DATA_BLOCK "DB_RecordData"   // DB70
{ S7_Optimized_Access := 'TRUE' }
// stored: AutoNumber false, MemoryReserve 100
   VAR
      xFP_ExportProdData { ExternalAccessible := 'False'; ExternalVisible := 'False'; ExternalWritable := 'False'} : Bool;
      xFP_ExportFlatCtrlRobot1 { ExternalAccessible := 'False'; ExternalVisible := 'False'; ExternalWritable := 'False'} : Bool;
      xFP_ExportFlatCtrlRobot2 { ExternalAccessible := 'False'; ExternalVisible := 'False'; ExternalWritable := 'False'} : Bool;
      xWriteDblExportProdDataBusy { ExternalAccessible := 'False'; ExternalVisible := 'False'; ExternalWritable := 'False'} : Bool;
      xWriteDblExportflatCtrlR1Busy { ExternalAccessible := 'False'; ExternalVisible := 'False'; ExternalWritable := 'False'} : Bool;
      xWriteDblExportFlatCtrlR2Busy { ExternalAccessible := 'False'; ExternalVisible := 'False'; ExternalWritable := 'False'} : Bool;
      nWriteDblExportProdDataResult { ExternalAccessible := 'False'; ExternalVisible := 'False'; ExternalWritable := 'False'} : Int;
      nWriteDblExportflatCtrlR1Result { ExternalAccessible := 'False'; ExternalVisible := 'False'; ExternalWritable := 'False'} : Int;
      nWriteDblExportFlatCtrlR2Result { ExternalAccessible := 'False'; ExternalVisible := 'False'; ExternalWritable := 'False'} : Int;
      xExportProdDataDone { ExternalAccessible := 'False'; ExternalVisible := 'False'; ExternalWritable := 'False'} : Bool;
      xExportProdDataBusy { ExternalAccessible := 'False'; ExternalVisible := 'False'; ExternalWritable := 'False'} : Bool;
      xExportProdDataError { ExternalAccessible := 'False'; ExternalVisible := 'False'; ExternalWritable := 'False'} : Bool;
      wExportProdDataStatus { ExternalAccessible := 'False'; ExternalVisible := 'False'; ExternalWritable := 'False'} : Word;
      wMemExportProdDataStatus { ExternalAccessible := 'False'; ExternalVisible := 'False'; ExternalWritable := 'False'} : Word;
      xExportFlatCtrlR1Done { ExternalAccessible := 'False'; ExternalVisible := 'False'; ExternalWritable := 'False'} : Bool;
      xExportFlatCtrlR1Busy { ExternalAccessible := 'False'; ExternalVisible := 'False'; ExternalWritable := 'False'} : Bool;
      xExportFlatCtrlR1Error { ExternalAccessible := 'False'; ExternalVisible := 'False'; ExternalWritable := 'False'} : Bool;
      wExportFlatCtrlR1Status { ExternalAccessible := 'False'; ExternalVisible := 'False'; ExternalWritable := 'False'} : Word;
      wMemExportFlatCtrlR1Status { ExternalAccessible := 'False'; ExternalVisible := 'False'; ExternalWritable := 'False'} : Word;
      xExportFlatCtrlR2Done { ExternalAccessible := 'False'; ExternalVisible := 'False'; ExternalWritable := 'False'} : Bool;
      xExportFlatCtrlR2Busy { ExternalAccessible := 'False'; ExternalVisible := 'False'; ExternalWritable := 'False'} : Bool;
      xExportFlatCtrlR2Error { ExternalAccessible := 'False'; ExternalVisible := 'False'; ExternalWritable := 'False'} : Bool;
      wExportFlatCtrlR2Status { ExternalAccessible := 'False'; ExternalVisible := 'False'; ExternalWritable := 'False'} : Word;
      wMemExportFlatCtrlR2Status { ExternalAccessible := 'False'; ExternalVisible := 'False'; ExternalWritable := 'False'} : Word;
   END_VAR
BEGIN
END_DATA_BLOCK

DATA_BLOCK "DBF_Safety"   // DB901, F_DB
{ S7_Optimized_Access := 'TRUE' }
// stored: AutoNumber false
   VAR
      TrueSafety { ExternalAccessible := 'False'; ExternalVisible := 'False'; ExternalWritable := 'False'} : Bool := TRUE;   // Safety Bool always TRUE
      FalseSafety { ExternalAccessible := 'False'; ExternalVisible := 'False'; ExternalWritable := 'False'} : Bool := FALSE;   // Safety Bool always FALSE
      Reset { ExternalAccessible := 'False'; ExternalVisible := 'False'; ExternalWritable := 'False'} : Bool;   // Reset bool
      ResetDoor { ExternalAccessible := 'False'; ExternalVisible := 'False'; ExternalWritable := 'False'} : Bool;   // Reset bool on maintenance door acces
      i_EStopOnMainCabinet { ExternalAccessible := 'False'; ExternalVisible := 'False'; ExternalWritable := 'False'} : Bool;   // Emergency stop state on main cabinet
      i_EStopLeftRopePull { ExternalAccessible := 'False'; ExternalVisible := 'False'; ExternalWritable := 'False'} : Bool;   // Emergency stop state rope pull left
      i_EStopRightRopePull { ExternalAccessible := 'False'; ExternalVisible := 'False'; ExternalWritable := 'False'} : Bool;   // Emergency stop state rope full right
      i_EStopEntryDoor { ExternalAccessible := 'False'; ExternalVisible := 'False'; ExternalWritable := 'False'} : Bool;   // Emergency stop state on entry guard locking
      i_DoorAcces { ExternalAccessible := 'False'; ExternalVisible := 'False'; ExternalWritable := 'False'} : Bool;   // Door state
      i_GateAccesCBS { ExternalAccessible := 'False'; ExternalVisible := 'False'; ExternalWritable := 'False'} : Bool;   // Gate acces state
      i_EStopControlRoom { ExternalAccessible := 'False'; ExternalVisible := 'False'; ExternalWritable := 'False'} : Bool;   // Emergency stop in the control room
      i_PedestrialDoorAcces { ExternalAccessible := 'False'; ExternalVisible := 'False'; ExternalWritable := 'False'} : Bool;   // Pedestrial door access state
      i_CaptiveKeyInLock { ExternalAccessible := 'False'; ExternalVisible := 'False'; ExternalWritable := 'False'} : Bool;   // Captive key on Lock
      i_EStopFromLeftRobot { ExternalAccessible := 'False'; ExternalVisible := 'False'; ExternalWritable := 'False'} : Bool;   // Emergency stop from flex pendant on the left robot
      i_EStopFromRightRobot { ExternalAccessible := 'False'; ExternalVisible := 'False'; ExternalWritable := 'False'} : Bool;   // Emergency stop from flex pendant on the right robot
      i_ReqEnableAirLeft { ExternalAccessible := 'False'; ExternalVisible := 'False'; ExternalWritable := 'False'} : Bool;   // Request enavle air pressure supply from left robot
      i_ReqEnableAirRight { ExternalAccessible := 'False'; ExternalVisible := 'False'; ExternalWritable := 'False'} : Bool;   // Request enavle air pressure supply from right robot
      i_RobotLeftStopped { ExternalAccessible := 'False'; ExternalVisible := 'False'; ExternalWritable := 'False'} : Bool;   // Left robot stooped
      i_RobotRightStopped { ExternalAccessible := 'False'; ExternalVisible := 'False'; ExternalWritable := 'False'} : Bool;   // Right robot stopped
      i_VacuumPumpRunning { ExternalAccessible := 'False'; ExternalVisible := 'False'; ExternalWritable := 'False'} : Bool;
      o_EnableAirSupplyLeftRobot { ExternalAccessible := 'False'; ExternalVisible := 'False'; ExternalWritable := 'False'} : Bool;   // Enable air pressure supply for left robot
      o_EnableAirSupplyRightRobot { ExternalAccessible := 'False'; ExternalVisible := 'False'; ExternalWritable := 'False'} : Bool;   // Enable air pressure supply for right robot
      o_EnableAirSupplySuctionUnit { ExternalAccessible := 'False'; ExternalVisible := 'False'; ExternalWritable := 'False'} : Bool;   // Enable air pressure supply for suction unit
      o_EStopSuctionUnit { ExternalAccessible := 'False'; ExternalVisible := 'False'; ExternalWritable := 'False'} : Bool;   // Emergency stop state to suction unit
      o_EStopToLeftRobot { ExternalAccessible := 'False'; ExternalVisible := 'False'; ExternalWritable := 'False'} : Bool;   // Cell emergency stop to left robot
      o_EStopToRightRobot { ExternalAccessible := 'False'; ExternalVisible := 'False'; ExternalWritable := 'False'} : Bool;   // Cell emergency stop to right robot
      o_OperatorProtectionToLeftRobot { ExternalAccessible := 'False'; ExternalVisible := 'False'; ExternalWritable := 'False'} : Bool;   // Operator protection state to the left robot
      o_OperatorProtectionToRightRobot { ExternalAccessible := 'False'; ExternalVisible := 'False'; ExternalWritable := 'False'} : Bool;   // Operator protection state to the right robot
      o_VacuumRunningDelayed { ExternalAccessible := 'False'; ExternalVisible := 'False'; ExternalWritable := 'False'} : Bool;   // Vacuum running delayed of
      l_GlobalEmergencyStopCell { ExternalAccessible := 'False'; ExternalVisible := 'False'; ExternalWritable := 'False'} : Bool;   // Global Emergency stop cell state
      l_GlobalEmergencyStop { ExternalAccessible := 'False'; ExternalVisible := 'False'; ExternalWritable := 'False'} : Bool;   // Global Emergency stop state
      l_GlobalEStopToLeftRobot { ExternalAccessible := 'False'; ExternalVisible := 'False'; ExternalWritable := 'False'} : Bool;   // Global Emergency stop state send to left robot
      l_GlobalEStopToRightRobot { ExternalAccessible := 'False'; ExternalVisible := 'False'; ExternalWritable := 'False'} : Bool;   // Global Emergency stop state send to right robot
      l_GlobalOperatorProtection { ExternalAccessible := 'False'; ExternalVisible := 'False'; ExternalWritable := 'False'} : Bool;   // Global door and gate state
      xErrorReadFromLeft { ExternalAccessible := 'False'; ExternalVisible := 'False'; ExternalWritable := 'False'} : Bool;
      xErrorReadFromRight { ExternalAccessible := 'False'; ExternalVisible := 'False'; ExternalWritable := 'False'} : Bool;
      xErrorWriteToLeft { ExternalAccessible := 'False'; ExternalVisible := 'False'; ExternalWritable := 'False'} : Bool;
      xErrorWriteToRight { ExternalAccessible := 'False'; ExternalVisible := 'False'; ExternalWritable := 'False'} : Bool;
      xAuthorStart { ExternalAccessible := 'False'; ExternalVisible := 'False'; ExternalWritable := 'False'} : Bool;
      xVacuumPumpRunning { ExternalAccessible := 'False'; ExternalVisible := 'False'; ExternalWritable := 'False'} : Bool;
   END_VAR
BEGIN
END_DATA_BLOCK

DATA_BLOCK "DB_FromSafety"   // DB998
{ S7_Optimized_Access := 'TRUE' }
// stored: AutoNumber false, MemoryReserve 100
   VAR
      EStopOnMainCabinet { ExternalAccessible := 'False'; ExternalVisible := 'False'; ExternalWritable := 'False'} : "stSafetyState";
      EstopLeftRopePull { ExternalAccessible := 'False'; ExternalVisible := 'False'; ExternalWritable := 'False'} : "stSafetyState";
      EstopRightRopePull { ExternalAccessible := 'False'; ExternalVisible := 'False'; ExternalWritable := 'False'} : "stSafetyState";
      EStopEntryDoor { ExternalAccessible := 'False'; ExternalVisible := 'False'; ExternalWritable := 'False'} : "stSafetyState";
      DoorAcces { ExternalAccessible := 'False'; ExternalVisible := 'False'; ExternalWritable := 'False'} : "stSafetyState";
      GateAccesCBS { ExternalAccessible := 'False'; ExternalVisible := 'False'; ExternalWritable := 'False'} : "stSafetyState";
      EStopControlRoom { ExternalAccessible := 'False'; ExternalVisible := 'False'; ExternalWritable := 'False'} : "stSafetyState";
      EnableAirSupplyLeftRobot { ExternalAccessible := 'False'; ExternalVisible := 'False'; ExternalWritable := 'False'} : "stSafetyState";
      EnableAirSupplyRightRobot { ExternalAccessible := 'False'; ExternalVisible := 'False'; ExternalWritable := 'False'} : "stSafetyState";
      EnableAirSupplySuctionUnit { ExternalAccessible := 'False'; ExternalVisible := 'False'; ExternalWritable := 'False'} : "stSafetyState";
      EStopSuctionUnit { ExternalAccessible := 'False'; ExternalVisible := 'False'; ExternalWritable := 'False'} : "stSafetyState";
      PedestrialDoorAcces { ExternalAccessible := 'False'; ExternalVisible := 'False'; ExternalWritable := 'False'} : "stSafetyState";
      CaptiveKeyInLock { ExternalAccessible := 'False'; ExternalVisible := 'False'; ExternalWritable := 'False'} : "stSafetyState";
      VacuumPumpRunning { ExternalAccessible := 'False'; ExternalVisible := 'False'; ExternalWritable := 'False'} : "stSafetyState";
      GlobalEStop { ExternalAccessible := 'False'; ExternalVisible := 'False'; ExternalWritable := 'False'; S7_SetPoint := 'True'} : "stSafetyState";
      xLeftRobotStopped { ExternalAccessible := 'False'; ExternalVisible := 'False'; ExternalWritable := 'False'} : Bool;
      xRightRobotStopped { ExternalAccessible := 'False'; ExternalVisible := 'False'; ExternalWritable := 'False'} : Bool;
      xEStopLeftRobot { ExternalAccessible := 'False'; ExternalVisible := 'False'; ExternalWritable := 'False'} : Bool;
      xEStopRightRobot { ExternalAccessible := 'False'; ExternalVisible := 'False'; ExternalWritable := 'False'} : Bool;
      xGlobalSafetyLeft { ExternalAccessible := 'False'; ExternalVisible := 'False'; ExternalWritable := 'False'} : Bool;
      xGlobalSafetyRight { ExternalAccessible := 'False'; ExternalVisible := 'False'; ExternalWritable := 'False'} : Bool;
      xAuthorStartVacuum { ExternalAccessible := 'False'; ExternalVisible := 'False'; ExternalWritable := 'False'} : Bool;
   END_VAR
BEGIN
END_DATA_BLOCK

DATA_BLOCK "DB_ToSafety"   // DB999
{ S7_Optimized_Access := 'TRUE' }
// stored: AutoNumber false, MemoryReserve 100
   VAR
      Reset { ExternalAccessible := 'False'; ExternalVisible := 'False'; ExternalWritable := 'False'} : Bool;   // Commande reset general
      ResetDoor { ExternalAccessible := 'False'; ExternalVisible := 'False'; ExternalWritable := 'False'} : Bool;   // Commande reset porte d'acces maintenance
      DoorLocked { ExternalAccessible := 'False'; ExternalVisible := 'False'; ExternalWritable := 'False'} : Bool;   // The door was locked
      VacuumDriveRunning { ExternalAccessible := 'False'; ExternalVisible := 'False'; ExternalWritable := 'False'} : Bool;   // Vacuum drive is running
      EnableVacuumRunning { ExternalAccessible := 'False'; ExternalVisible := 'False'; ExternalWritable := 'False'} : Bool;   // Enable vacuum running
   END_VAR
BEGIN
END_DATA_BLOCK

ORGANIZATION_BLOCK "Main"   // OB1, LAD, ProgramCycle
TITLE = "Main Program Sweep (Cycle)"
{ S7_Optimized_Access := 'TRUE' }
// stored: SetENOAutomatically false
   VAR_INPUT
      Initial_Call : Bool;   // Initial call of this OB
      Remanence : Bool;   // =True, if remanent data are available
   END_VAR
BEGIN

REGION Network 1
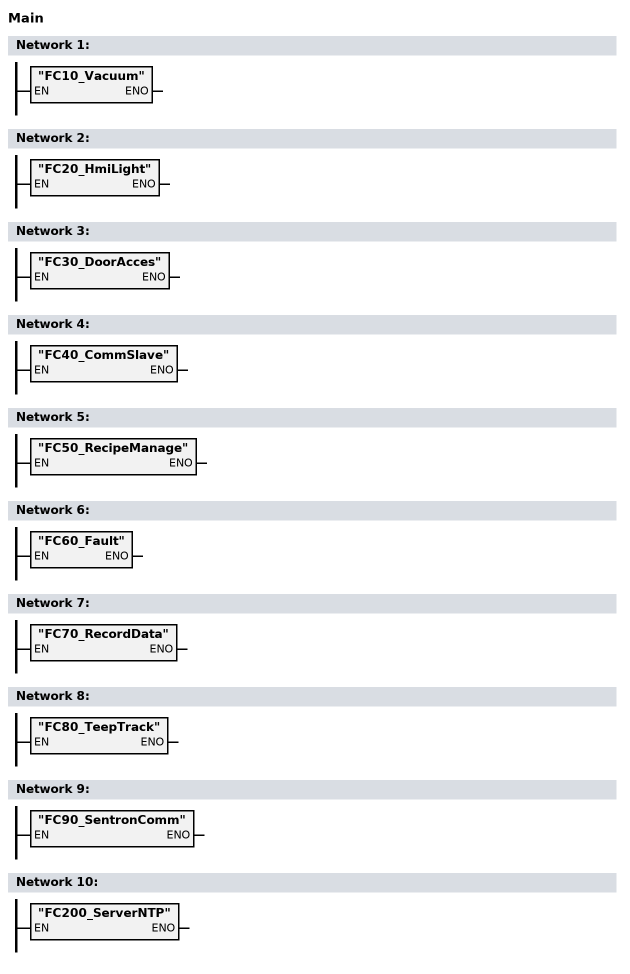
   RUNG wire#powerrail
      "FC10_Vacuum"()
   END_RUNG
   // the same network as SCL:
   "FC10_Vacuum"();
END_REGION

REGION Network 2
   RUNG wire#powerrail
      "FC20_HmiLight"()
   END_RUNG
   // the same network as SCL:
   "FC20_HmiLight"();
END_REGION

REGION Network 3
   RUNG wire#powerrail
      "FC30_DoorAcces"()
   END_RUNG
   // the same network as SCL:
   "FC30_DoorAcces"();
END_REGION

REGION Network 4
   RUNG wire#powerrail
      "FC40_CommSlave"()
   END_RUNG
   // the same network as SCL:
   "FC40_CommSlave"();
END_REGION

REGION Network 5
   RUNG wire#powerrail
      "FC50_RecipeManage"()
   END_RUNG
   // the same network as SCL:
   "FC50_RecipeManage"();
END_REGION

REGION Network 6
   RUNG wire#powerrail
      "FC60_Fault"()
   END_RUNG
   // the same network as SCL:
   "FC60_Fault"();
END_REGION

REGION Network 7
   RUNG wire#powerrail
      "FC70_RecordData"()
   END_RUNG
   // the same network as SCL:
   "FC70_RecordData"();
END_REGION

REGION Network 8
   RUNG wire#powerrail
      "FC80_TeepTrack"()
   END_RUNG
   // the same network as SCL:
   "FC80_TeepTrack"();
END_REGION

REGION Network 9
   RUNG wire#powerrail
      "FC90_SentronComm"()
   END_RUNG
   // the same network as SCL:
   "FC90_SentronComm"();
END_REGION

REGION Network 10
   RUNG wire#powerrail
      "FC200_ServerNTP"()
   END_RUNG
   // the same network as SCL:
   "FC200_ServerNTP"();
END_REGION
END_ORGANIZATION_BLOCK

FUNCTION "FC10_Vacuum" : Void   // FC10, LAD
{ S7_Optimized_Access := 'TRUE' }
// stored: AutoNumber false, IsIECCheckEnabled true, SetENOAutomatically false
BEGIN

REGION Network 1: Complet management of Vacuum system
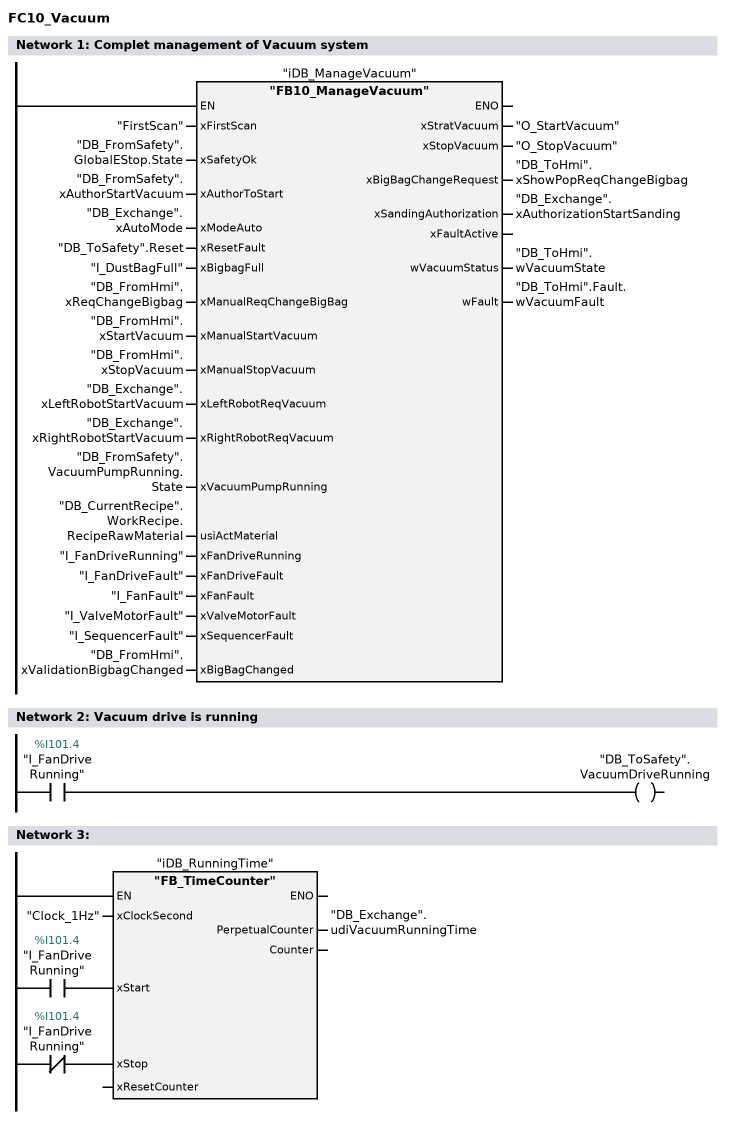
   RUNG wire#powerrail
      "iDB_ManageVacuum"(xFirstScan := "FirstScan", xSafetyOk := "DB_FromSafety".GlobalEStop.State, xAuthorToStart := "DB_FromSafety".xAuthorStartVacuum, xModeAuto := "DB_Exchange".xAutoMode, xResetFault := "DB_ToSafety".Reset, xBigbagFull := "I_DustBagFull", xManualReqChangeBigBag := "DB_FromHmi".xReqChangeBigbag, xManualStartVacuum := "DB_FromHmi".xStartVacuum, xManualStopVacuum := "DB_FromHmi".xStopVacuum, xLeftRobotReqVacuum := "DB_Exchange".xLeftRobotStartVacuum, xRightRobotReqVacuum := "DB_Exchange".xRightRobotStartVacuum, xVacuumPumpRunning := "DB_FromSafety".VacuumPumpRunning.State, usiActMaterial := "DB_CurrentRecipe".WorkRecipe.RecipeRawMaterial, xFanDriveRunning := "I_FanDriveRunning", xFanDriveFault := "I_FanDriveFault", xFanFault := "I_FanFault", xValveMotorFault := "I_ValveMotorFault", xSequencerFault := "I_SequencerFault", xBigBagChanged := "DB_FromHmi".xValidationBigbagChanged, xStratVacuum => "O_StartVacuum", xStopVacuum => "O_StopVacuum", xBigBagChangeRequest => "DB_ToHmi".xShowPopReqChangeBigbag, xSandingAuthorization => "DB_Exchange".xAuthorizationStartSanding, xFaultActive =>, wVacuumStatus => "DB_ToHmi".wVacuumState, wFault => "DB_ToHmi".Fault.wVacuumFault)
   END_RUNG
   // the same network as SCL:
   "iDB_ManageVacuum"(xFirstScan := "FirstScan",   // "FB10_ManageVacuum"
                      xSafetyOk := "DB_FromSafety".GlobalEStop.State,
                      xAuthorToStart := "DB_FromSafety".xAuthorStartVacuum,
                      xModeAuto := "DB_Exchange".xAutoMode,
                      xResetFault := "DB_ToSafety".Reset,
                      xBigbagFull := "I_DustBagFull",
                      xManualReqChangeBigBag := "DB_FromHmi".xReqChangeBigbag,
                      xManualStartVacuum := "DB_FromHmi".xStartVacuum,
                      xManualStopVacuum := "DB_FromHmi".xStopVacuum,
                      xLeftRobotReqVacuum := "DB_Exchange".xLeftRobotStartVacuum,
                      xRightRobotReqVacuum := "DB_Exchange".xRightRobotStartVacuum,
                      xVacuumPumpRunning := "DB_FromSafety".VacuumPumpRunning.State,
                      usiActMaterial := "DB_CurrentRecipe".WorkRecipe.RecipeRawMaterial,
                      xFanDriveRunning := "I_FanDriveRunning",
                      xFanDriveFault := "I_FanDriveFault",
                      xFanFault := "I_FanFault",
                      xValveMotorFault := "I_ValveMotorFault",
                      xSequencerFault := "I_SequencerFault",
                      xBigBagChanged := "DB_FromHmi".xValidationBigbagChanged,
                      xStratVacuum => "O_StartVacuum",
                      xStopVacuum => "O_StopVacuum",
                      xBigBagChangeRequest => "DB_ToHmi".xShowPopReqChangeBigbag,
                      xSandingAuthorization => "DB_Exchange".xAuthorizationStartSanding,
                      wVacuumStatus => "DB_ToHmi".wVacuumState,
                      wFault => "DB_ToHmi".Fault.wVacuumFault);
END_REGION

REGION Network 2: Vacuum drive is running
   RUNG wire#powerrail
      Contact( "I_FanDriveRunning" )
      Coil( "DB_ToSafety".VacuumDriveRunning )
   END_RUNG
   // the same network as SCL:
   "DB_ToSafety".VacuumDriveRunning := "I_FanDriveRunning";
END_REGION

REGION Network 3
   RUNG wire#powerrail
      "iDB_RunningTime"(xStart := wire#w1, xStop := wire#w2, xClockSecond := "Clock_1Hz", xResetCounter :=, PerpetualCounter => "DB_Exchange".udiVacuumRunningTime, "Counter" =>)
   END_RUNG
   RUNG wire#powerrail
      Contact( "I_FanDriveRunning" )
   END_RUNG wire#w1
   RUNG wire#powerrail
      I_Contact( "I_FanDriveRunning" )
   END_RUNG wire#w2
   // the same network as SCL:
   "iDB_RunningTime"(xClockSecond := "Clock_1Hz",   // "FB_TimeCounter"
                     xStart := "I_FanDriveRunning",
                     xStop := NOT "I_FanDriveRunning",
                     PerpetualCounter => "DB_Exchange".udiVacuumRunningTime);
END_REGION
END_FUNCTION

FUNCTION_BLOCK "FB10_ManageVacuum"   // FB10, LAD
{ S7_Optimized_Access := 'TRUE' }
// stored: AutoNumber false, IsIECCheckEnabled true, MemoryReserve 100, SetENOAutomatically true
   VAR_INPUT
      xFirstScan { ExternalAccessible := 'False'; ExternalVisible := 'False'; ExternalWritable := 'False'} : Bool;
      xSafetyOk { ExternalAccessible := 'False'; ExternalVisible := 'False'; ExternalWritable := 'False'} : Bool;   // General Safety state
      xAuthorToStart { ExternalAccessible := 'False'; ExternalVisible := 'False'; ExternalWritable := 'False'} : Bool;   // Authorisation to start Vacuum
      xModeAuto { ExternalAccessible := 'False'; ExternalVisible := 'False'; ExternalWritable := 'False'} : Bool;   // Mode auto active
      xResetFault { ExternalAccessible := 'False'; ExternalVisible := 'False'; ExternalWritable := 'False'} : Bool;   // Reset fault
      xBigbagFull { ExternalAccessible := 'False'; ExternalVisible := 'False'; ExternalWritable := 'False'} : Bool;   // Big Bag is full
      xManualReqChangeBigBag { ExternalAccessible := 'False'; ExternalVisible := 'False'; ExternalWritable := 'False'} : Bool;   // Manual request changing Big bag
      xManualStartVacuum { ExternalAccessible := 'False'; ExternalVisible := 'False'; ExternalWritable := 'False'} : Bool;   // Manual enabling Vacuum
      xManualStopVacuum { ExternalAccessible := 'False'; ExternalVisible := 'False'; ExternalWritable := 'False'} : Bool;   // Manual stopping Vacuum
      xLeftRobotReqVacuum { ExternalAccessible := 'False'; ExternalVisible := 'False'; ExternalWritable := 'False'} : Bool;   // Left Robot request enabling Vacuum
      xRightRobotReqVacuum { ExternalAccessible := 'False'; ExternalVisible := 'False'; ExternalWritable := 'False'} : Bool;   // Right Robot request enabling Vacuum
      xVacuumPumpRunning { ExternalAccessible := 'False'; ExternalVisible := 'False'; ExternalWritable := 'False'} : Bool;   // Vacuum Pump Running
      usiActMaterial { ExternalAccessible := 'False'; ExternalVisible := 'False'; ExternalWritable := 'False'} : USInt;   // Type of material for actual production
      xFanDriveRunning { ExternalAccessible := 'False'; ExternalVisible := 'False'; ExternalWritable := 'False'} : Bool;   // State fan drive running
      xFanDriveFault { ExternalAccessible := 'False'; ExternalVisible := 'False'; ExternalWritable := 'False'} : Bool;   // fault fan drive
      xFanFault { ExternalAccessible := 'False'; ExternalVisible := 'False'; ExternalWritable := 'False'} : Bool;   // Fault fan
      xValveMotorFault { ExternalAccessible := 'False'; ExternalVisible := 'False'; ExternalWritable := 'False'} : Bool;   // Fault Valve motor
      xSequencerFault { ExternalAccessible := 'False'; ExternalVisible := 'False'; ExternalWritable := 'False'} : Bool;   // Fault sequencer
   END_VAR
   VAR_OUTPUT
      xStratVacuum { ExternalAccessible := 'False'; ExternalVisible := 'False'; ExternalWritable := 'False'} : Bool;   // Start Vacuum
      xStopVacuum { ExternalAccessible := 'False'; ExternalVisible := 'False'; ExternalWritable := 'False'} : Bool;   // Stop Vacuum
      xBigBagChangeRequest { ExternalAccessible := 'False'; ExternalVisible := 'False'; ExternalWritable := 'False'} : Bool;   // Big Bag change request
      xSandingAuthorization { ExternalAccessible := 'False'; ExternalVisible := 'False'; ExternalWritable := 'False'} : Bool;   // Sanding authorisation
      xFaultActive { ExternalAccessible := 'False'; ExternalVisible := 'False'; ExternalWritable := 'False'} : Bool;
      wVacuumStatus { ExternalAccessible := 'False'; ExternalVisible := 'False'; ExternalWritable := 'False'} : Word;   // Vacuum Status for HMI
      wFault { ExternalAccessible := 'False'; ExternalVisible := 'False'; ExternalWritable := 'False'} : Word;   // Fault number
   END_VAR
   VAR_IN_OUT
      xBigBagChanged { ExternalAccessible := 'False'; ExternalVisible := 'False'; ExternalWritable := 'False'} : Bool;   // Validation operator Big Bag changed
   END_VAR
   VAR
      sxBigBagChangeReq { ExternalAccessible := 'False'; ExternalVisible := 'False'; ExternalWritable := 'False'} : Bool;
      sxVacuumAuto { ExternalAccessible := 'False'; ExternalVisible := 'False'; ExternalWritable := 'False'} : Bool;
      sxVacuumManual { ExternalAccessible := 'False'; ExternalVisible := 'False'; ExternalWritable := 'False'} : Bool;
      sxToggleAuto { ExternalAccessible := 'False'; ExternalVisible := 'False'; ExternalWritable := 'False'} : Bool;
   END_VAR
   VAR RETAIN
      susiPrevMaterial { ExternalAccessible := 'False'; ExternalVisible := 'False'; ExternalWritable := 'False'} : USInt;   // Type of material for previus production
   END_VAR
   VAR
      suiStep { ExternalAccessible := 'False'; ExternalVisible := 'False'; ExternalWritable := 'False'} : UInt;
      miDB_RobotReqVacuum { ExternalAccessible := 'False'; ExternalVisible := 'False'; ExternalWritable := 'False'; S7_SetPoint := 'True'} : TOF_TIME;
      miDB_TonAuthorToStart { ExternalAccessible := 'False'; ExternalVisible := 'False'; ExternalWritable := 'False'; S7_SetPoint := 'True'} : TON_TIME;
      miDB_TonSetp10 { ExternalAccessible := 'False'; ExternalVisible := 'False'; ExternalWritable := 'False'; S7_SetPoint := 'True'} : TON_TIME;
   END_VAR
   VAR CONSTANT
      cuiInitialStep : UInt := 0;
      cuiWaitBigBagChanged : UInt := 5;
      cuiWaitStartVacuum : UInt := 10;
      cuiRunVacuum : UInt := 15;
      cuiWaitStopVacuum : UInt := 20;
      cuiStopVacuum : UInt := 25;
   END_VAR
BEGIN

REGION Network 1 (SCL): Fault number
   // Reset fault
   IF #xResetFault THEN
     #wFault := 16#0;
   END_IF;

   // Sequencer fault
   IF NOT #xSequencerFault THEN
     #wFault.%X0 := TRUE;
   END_IF;

   // Fan drive fault
   IF #xFanDriveFault THEN
     #wFault.%X1 := TRUE;
   END_IF;

   // Breaker 11Q1 in AER cabinet fault
   IF #xFanFault AND (NOT #xFanDriveFault) THEN
     #wFault.%X2 := TRUE;
   END_IF;

   // Breaker 10Q1 in AER cabinet fault
   IF #xValveMotorFault THEN
     #wFault.%X3 := TRUE;
   END_IF;

   #miDB_TonAuthorToStart(IN:=(NOT #xFanDriveRunning) AND (NOT #xAuthorToStart),
                          PT:=T#10S);
   IF #miDB_TonAuthorToStart.Q THEN
     #wFault.%X4 := TRUE;
   END_IF;

   // At least one active fault
   #xFaultActive := (#wFault <> 16#0);
END_REGION

REGION Network 2: At least one robot request vacumm
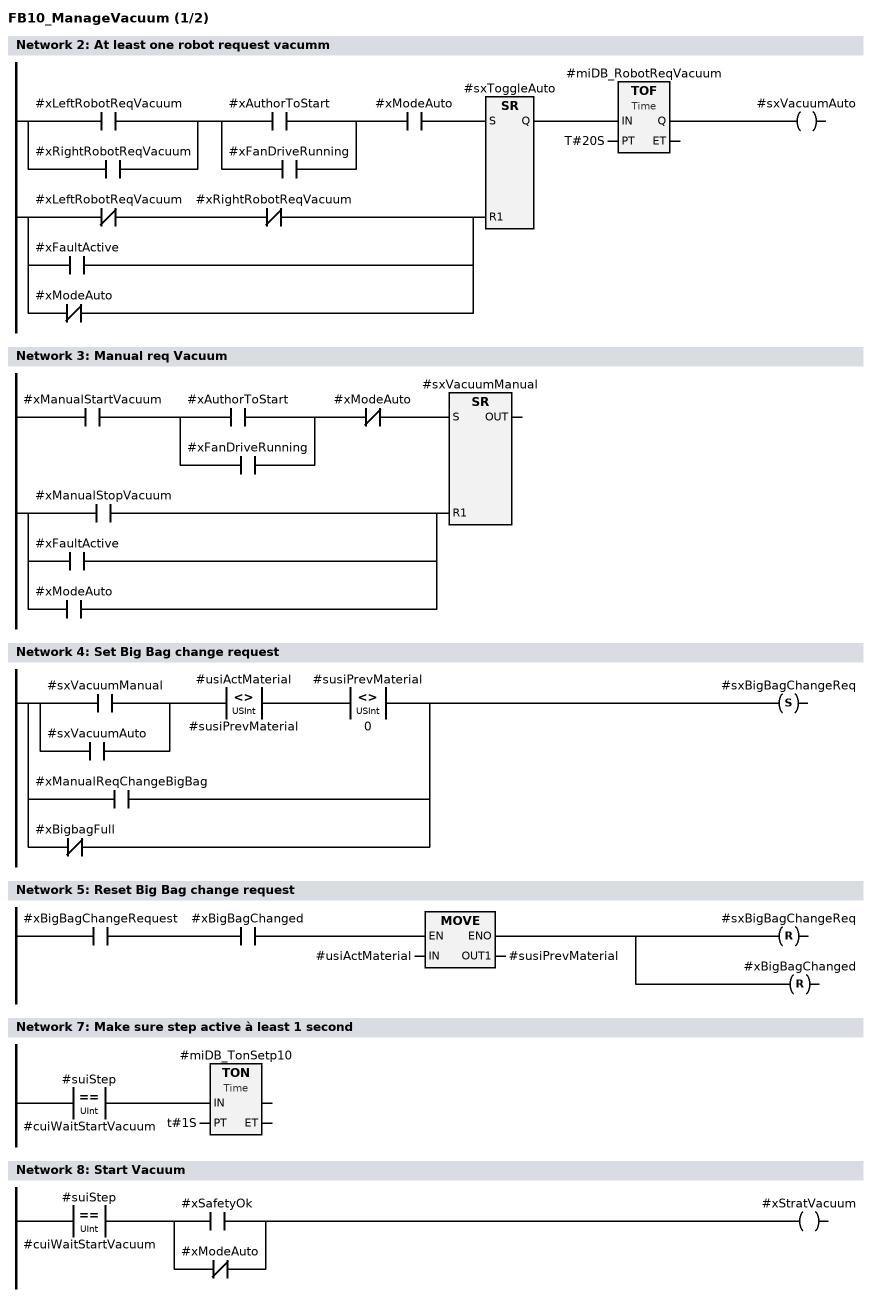
   RUNG wire#powerrail
      Contact( #xLeftRobotReqVacuum )
      wire#w1
      Contact( #xAuthorToStart )
      wire#w2
      Contact( #xModeAuto )
      S_SR(operand := #sxToggleAuto, r1 := wire#w3)
      { S7_Templates := "time_type := Time" } #miDB_RobotReqVacuum.TOF(pt := T#20S, et =>)
      Coil( #sxVacuumAuto )
   END_RUNG
   RUNG wire#powerrail
      Contact( #xRightRobotReqVacuum )
   END_RUNG wire#w1
   RUNG wire#w1
      Contact( #xFanDriveRunning )
   END_RUNG wire#w2
   RUNG wire#powerrail
      I_Contact( #xLeftRobotReqVacuum )
      I_Contact( #xRightRobotReqVacuum )
   END_RUNG wire#w3
   RUNG wire#powerrail
      Contact( #xFaultActive )
   END_RUNG wire#w3
   RUNG wire#powerrail
      I_Contact( #xModeAuto )
   END_RUNG wire#w3
   // the same network as SCL:
   IF (#xLeftRobotReqVacuum OR #xRightRobotReqVacuum) AND (#xAuthorToStart OR #xFanDriveRunning) AND #xModeAuto THEN
       #sxToggleAuto := TRUE;   // SR flip-flop
   END_IF;
   IF (NOT #xLeftRobotReqVacuum AND NOT #xRightRobotReqVacuum) OR #xFaultActive OR NOT #xModeAuto THEN
       #sxToggleAuto := FALSE;
   END_IF;
   #miDB_RobotReqVacuum(IN := #sxToggleAuto, PT := T#20S);   // TOF
   #sxVacuumAuto := #miDB_RobotReqVacuum.Q;
END_REGION

REGION Network 3: Manual req Vacuum
   RUNG wire#powerrail
      Contact( #xManualStartVacuum )
      wire#w1
      Contact( #xAuthorToStart )
      wire#w2
      I_Contact( #xModeAuto )
      S_SR(operand := #sxVacuumManual, r1 := wire#w3)
   END_RUNG
   RUNG wire#w1
      Contact( #xFanDriveRunning )
   END_RUNG wire#w2
   RUNG wire#powerrail
      Contact( #xManualStopVacuum )
   END_RUNG wire#w3
   RUNG wire#powerrail
      Contact( #xFaultActive )
   END_RUNG wire#w3
   RUNG wire#powerrail
      Contact( #xModeAuto )
   END_RUNG wire#w3
   // the same network as SCL:
   IF #xManualStartVacuum AND (#xAuthorToStart OR #xFanDriveRunning) AND NOT #xModeAuto THEN
       #sxVacuumManual := TRUE;   // SR flip-flop
   END_IF;
   IF #xManualStopVacuum OR #xFaultActive OR #xModeAuto THEN #sxVacuumManual := FALSE; END_IF;
END_REGION

REGION Network 4: Set Big Bag change request
   RUNG wire#powerrail
      Contact( #sxVacuumManual )
      wire#w1
      { S7_Templates := "SrcType := USInt" } NE_Contact(in1 := #usiActMaterial, in2 := #susiPrevMaterial)
      { S7_Templates := "SrcType := USInt" } NE_Contact(in1 := #susiPrevMaterial, in2 := 0)
      wire#w2
      S_Coil( #sxBigBagChangeReq )
   END_RUNG
   RUNG wire#powerrail
      Contact( #sxVacuumAuto )
   END_RUNG wire#w1
   RUNG wire#powerrail
      Contact( #xManualReqChangeBigBag )
   END_RUNG wire#w2
   RUNG wire#powerrail
      I_Contact( #xBigbagFull )
   END_RUNG wire#w2
   // the same network as SCL:
   IF ((#sxVacuumManual OR #sxVacuumAuto) AND (#usiActMaterial <> #susiPrevMaterial) AND (#susiPrevMaterial <> 0)) OR #xManualReqChangeBigBag OR NOT #xBigbagFull THEN
       #sxBigBagChangeReq := TRUE;
   END_IF;
END_REGION

REGION Network 5: Reset Big Bag change request
   RUNG wire#powerrail
      Contact( #xBigBagChangeRequest )
      Contact( #xBigBagChanged )
      Move(in := #usiActMaterial, out1 => #susiPrevMaterial)
      wire#w1
      R_Coil( #sxBigBagChangeReq )
   END_RUNG
   RUNG wire#w1
      R_Coil( #xBigBagChanged )
   END_RUNG
   // the same network as SCL:
   IF #xBigBagChangeRequest AND #xBigBagChanged THEN
       #susiPrevMaterial := #usiActMaterial;
       #sxBigBagChangeReq := FALSE;
       #xBigBagChanged := FALSE;
   END_IF;
END_REGION

REGION Network 6 (SCL): Sequencer Vacuum
   // Initialise sequence at first scan of PLC
   IF #xFirstScan THEN
     #suiStep := #cuiInitialStep;
   END_IF;

   // Sequencer step
   CASE #suiStep OF
     #cuiInitialStep:
       IF (#sxVacuumAuto OR #sxVacuumManual) AND #xSafetyOk AND (NOT #sxBigBagChangeReq) THEN
         #suiStep := #cuiWaitStartVacuum;
       ELSIF (#sxVacuumAuto OR #sxVacuumManual) AND #xSafetyOk AND #sxBigBagChangeReq THEN
         #suiStep := #cuiWaitBigBagChanged;
       END_IF;

     #cuiWaitBigBagChanged:
       IF (NOT #sxBigBagChangeReq) THEN
         #suiStep := #cuiWaitStartVacuum;
       END_IF;

     #cuiWaitStartVacuum:
       IF #xFanDriveRunning AND #miDB_TonSetp10.Q THEN
         #suiStep := #cuiRunVacuum;
       END_IF;

     #cuiRunVacuum:
       IF ((NOT #sxVacuumAuto) AND (NOT #sxVacuumManual)) OR (NOT #xSafetyOk) THEN
         #suiStep := #cuiWaitStopVacuum;
       END_IF;

     #cuiWaitStopVacuum:
       IF (NOT #xFanDriveRunning) THEN
         #suiStep := #cuiStopVacuum;
       ELSIF (#sxVacuumAuto OR #sxVacuumManual) AND #xSafetyOk THEN
         #suiStep := #cuiWaitStartVacuum;
       END_IF;

     #cuiStopVacuum:
       IF #xAuthorToStart THEN;
         #suiStep := #cuiInitialStep;
       END_IF;

     ELSE  // Statement section ELSE
       // Error in this case
       ;
   END_CASE;
END_REGION

REGION Network 7: Make sure step active à least 1 second
   RUNG wire#powerrail
      { S7_Templates := "SrcType := UInt" } EQ_Contact(in1 := #suiStep, in2 := #cuiWaitStartVacuum)
      { S7_Templates := "time_type := Time" } #miDB_TonSetp10.TON(pt := t#1S, et =>)
   END_RUNG
   // the same network as SCL:
   #miDB_TonSetp10(IN := #suiStep = #cuiWaitStartVacuum, PT := t#1S);   // TON
END_REGION

REGION Network 8: Start Vacuum
   RUNG wire#powerrail
      { S7_Templates := "SrcType := UInt" } EQ_Contact(in1 := #suiStep, in2 := #cuiWaitStartVacuum)
      wire#w1
      Contact( #xSafetyOk )
      wire#w2
      Coil( #xStratVacuum )
   END_RUNG
   RUNG wire#w1
      I_Contact( #xModeAuto )
   END_RUNG wire#w2
   // the same network as SCL:
   #xStratVacuum := (#suiStep = #cuiWaitStartVacuum) AND (#xSafetyOk OR NOT #xModeAuto);
END_REGION

REGION Network 9: Stop Vacuum
   // Shunt a enlever
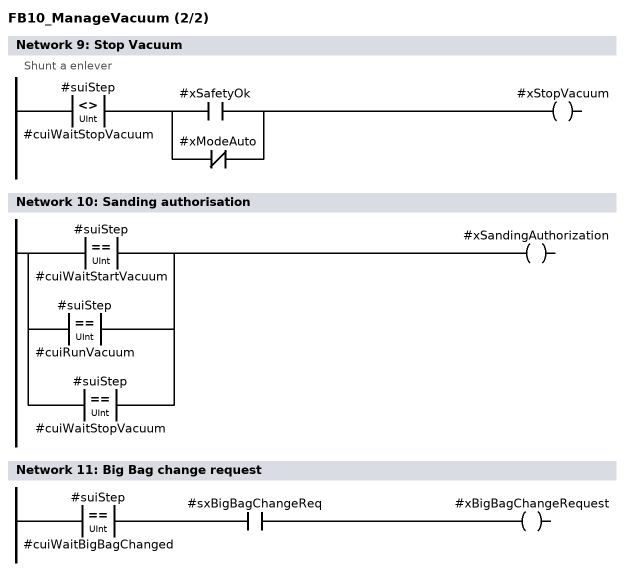
   RUNG wire#powerrail
      { S7_Templates := "SrcType := UInt" } NE_Contact(in1 := #suiStep, in2 := #cuiWaitStopVacuum)
      wire#w1
      Contact( #xSafetyOk )
      wire#w2
      Coil( #xStopVacuum )
   END_RUNG
   RUNG wire#w1
      I_Contact( #xModeAuto )
   END_RUNG wire#w2
   // the same network as SCL:
   #xStopVacuum := (#suiStep <> #cuiWaitStopVacuum) AND (#xSafetyOk OR NOT #xModeAuto);
END_REGION

REGION Network 10: Sanding authorisation
   RUNG wire#powerrail
      { S7_Templates := "SrcType := UInt" } EQ_Contact(in1 := #suiStep, in2 := #cuiWaitStartVacuum)
      wire#w1
      Coil( #xSandingAuthorization )
   END_RUNG
   RUNG wire#powerrail
      { S7_Templates := "SrcType := UInt" } EQ_Contact(in1 := #suiStep, in2 := #cuiRunVacuum)
   END_RUNG wire#w1
   RUNG wire#powerrail
      { S7_Templates := "SrcType := UInt" } EQ_Contact(in1 := #suiStep, in2 := #cuiWaitStopVacuum)
   END_RUNG wire#w1
   // the same network as SCL:
   #xSandingAuthorization := (#suiStep = #cuiWaitStartVacuum) OR (#suiStep = #cuiRunVacuum) OR (#suiStep = #cuiWaitStopVacuum);
END_REGION

REGION Network 11: Big Bag change request
   RUNG wire#powerrail
      { S7_Templates := "SrcType := UInt" } EQ_Contact(in1 := #suiStep, in2 := #cuiWaitBigBagChanged)
      Contact( #sxBigBagChangeReq )
      Coil( #xBigBagChangeRequest )
   END_RUNG
   // the same network as SCL:
   #xBigBagChangeRequest := (#suiStep = #cuiWaitBigBagChanged) AND #sxBigBagChangeReq;
END_REGION

REGION Network 12 (SCL): Vacuum Status
   // Reset Vacuum Status
   #wVacuumStatus := 16#0;
   // If Fault set bit 1
   IF #xFaultActive THEN // Show at list one fault active
     #wVacuumStatus := 16#1;
   ELSIF (NOT #xBigbagFull) THEN // Big Bag Full
     #wVacuumStatus := 16#2;
   ELSE
     // Fan drive activated
     IF #xFanDriveRunning THEN
       #wVacuumStatus := #wVacuumStatus OR 16#4;
     END_IF;

     // VacuumPump running
     IF #xVacuumPumpRunning THEN
       #wVacuumStatus := #wVacuumStatus OR 16#8;
     END_IF;

     CASE #suiStep OF

       #cuiInitialStep:
         #wVacuumStatus := #wVacuumStatus OR 16#10;

       #cuiWaitBigBagChanged:
         #wVacuumStatus := #wVacuumStatus OR 16#20;

       #cuiWaitStartVacuum, #cuiRunVacuum:
         #wVacuumStatus := #wVacuumStatus OR 16#40;

       #cuiWaitStopVacuum, #cuiStopVacuum:
         #wVacuumStatus := #wVacuumStatus OR 16#80;

     END_CASE;
   END_IF;
END_REGION
END_FUNCTION_BLOCK

FUNCTION "FC20_HmiLight" : Void   // FC20, LAD
{ S7_Optimized_Access := 'TRUE' }
// stored: AutoNumber false, IsIECCheckEnabled true, SetENOAutomatically false
   VAR_TEMP
      txStartUpWarning : Bool;
      txFaultError : Bool;
      txConditionOk : Bool;
      txReqOperator : Bool;
   END_VAR
   VAR CONSTANT
      cusiAutoMode : USInt := 1;   // Automatic mode
      cusiSemiAutoMode : USInt := 3;   // Semi-Automatic mode
      cusiMaintenanceMode : USInt := 2;   // Maintenance mode
   END_VAR
   VAR_TEMP   // added for the SCL form of the ladder/FBD networks
      _w1 : Bool;
      _w2 : Bool;
   END_VAR
BEGIN

REGION Network 1: Commande reset general
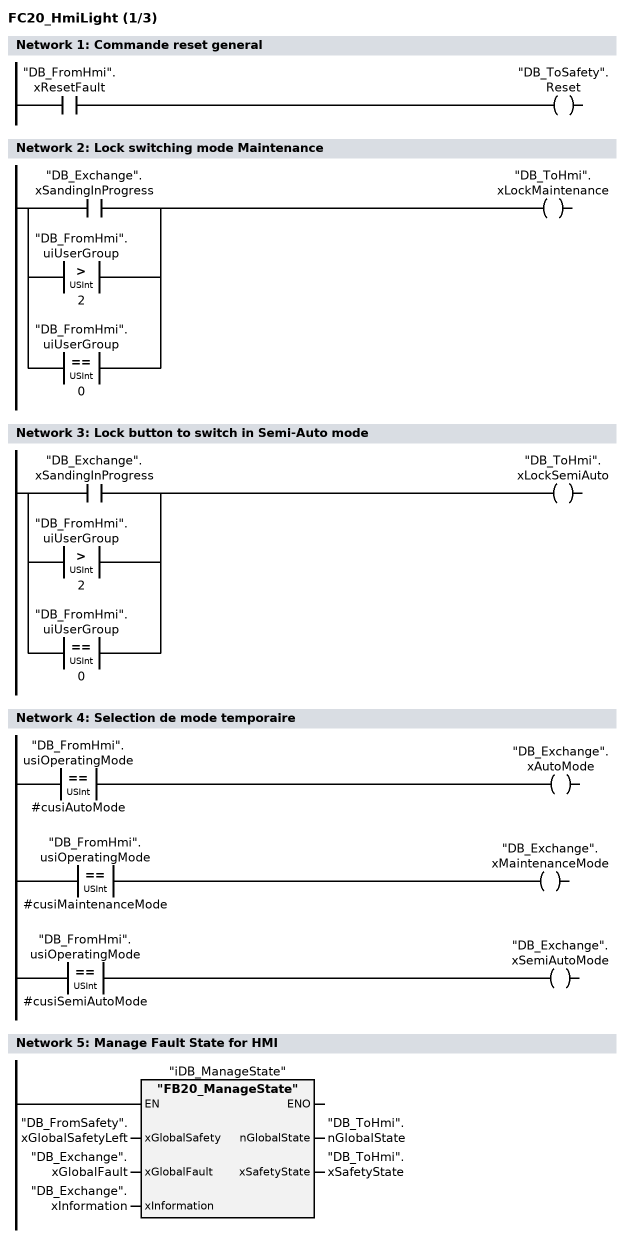
   RUNG wire#powerrail
      Contact( "DB_FromHmi".xResetFault )
      Coil( "DB_ToSafety".Reset )
   END_RUNG
   // the same network as SCL:
   "DB_ToSafety".Reset := "DB_FromHmi".xResetFault;
END_REGION

REGION Network 2: Lock switching mode Maintenance
   RUNG wire#powerrail
      Contact( "DB_Exchange".xSandingInProgress )
      wire#w1
      Coil( "DB_ToHmi".xLockMaintenance )
   END_RUNG
   RUNG wire#powerrail
      { S7_Templates := "SrcType := USInt" } GT_Contact(in1 := "DB_FromHmi".uiUserGroup, in2 := 2)
   END_RUNG wire#w1
   RUNG wire#powerrail
      { S7_Templates := "SrcType := USInt" } EQ_Contact(in1 := "DB_FromHmi".uiUserGroup, in2 := 0)
   END_RUNG wire#w1
   // the same network as SCL:
   "DB_ToHmi".xLockMaintenance := "DB_Exchange".xSandingInProgress OR ("DB_FromHmi".uiUserGroup > 2) OR ("DB_FromHmi".uiUserGroup = 0);
END_REGION

REGION Network 3: Lock button to switch in Semi-Auto mode
   RUNG wire#powerrail
      Contact( "DB_Exchange".xSandingInProgress )
      wire#w1
      Coil( "DB_ToHmi".xLockSemiAuto )
   END_RUNG
   RUNG wire#powerrail
      { S7_Templates := "SrcType := USInt" } GT_Contact(in1 := "DB_FromHmi".uiUserGroup, in2 := 2)
   END_RUNG wire#w1
   RUNG wire#powerrail
      { S7_Templates := "SrcType := USInt" } EQ_Contact(in1 := "DB_FromHmi".uiUserGroup, in2 := 0)
   END_RUNG wire#w1
   // the same network as SCL:
   "DB_ToHmi".xLockSemiAuto := "DB_Exchange".xSandingInProgress OR ("DB_FromHmi".uiUserGroup > 2) OR ("DB_FromHmi".uiUserGroup = 0);
END_REGION

REGION Network 4: Selection de mode temporaire
   RUNG wire#powerrail
      { S7_Templates := "SrcType := USInt" } EQ_Contact(in1 := "DB_FromHmi".usiOperatingMode, in2 := #cusiAutoMode)
      Coil( "DB_Exchange".xAutoMode )
   END_RUNG
   RUNG wire#powerrail
      { S7_Templates := "SrcType := USInt" } EQ_Contact(in1 := "DB_FromHmi".usiOperatingMode, in2 := #cusiMaintenanceMode)
      Coil( "DB_Exchange".xMaintenanceMode )
   END_RUNG
   RUNG wire#powerrail
      { S7_Templates := "SrcType := USInt" } EQ_Contact(in1 := "DB_FromHmi".usiOperatingMode, in2 := #cusiSemiAutoMode)
      Coil( "DB_Exchange".xSemiAutoMode )
   END_RUNG
   // the same network as SCL:
   "DB_Exchange".xAutoMode := "DB_FromHmi".usiOperatingMode = #cusiAutoMode;
   "DB_Exchange".xMaintenanceMode := "DB_FromHmi".usiOperatingMode = #cusiMaintenanceMode;
   "DB_Exchange".xSemiAutoMode := "DB_FromHmi".usiOperatingMode = #cusiSemiAutoMode;
END_REGION

REGION Network 5: Manage Fault State for HMI
   RUNG wire#powerrail
      "iDB_ManageState"(xGlobalSafety := "DB_FromSafety".xGlobalSafetyLeft, xGlobalFault := "DB_Exchange".xGlobalFault, xInformation := "DB_Exchange".xInformation, nGlobalState => "DB_ToHmi".nGlobalState, xSafetyState => "DB_ToHmi".xSafetyState)
   END_RUNG
   // the same network as SCL:
   "iDB_ManageState"(xGlobalSafety := "DB_FromSafety".xGlobalSafetyLeft,   // "FB20_ManageState"
                     xGlobalFault := "DB_Exchange".xGlobalFault,
                     xInformation := "DB_Exchange".xInformation,
                     nGlobalState => "DB_ToHmi".nGlobalState,
                     xSafetyState => "DB_ToHmi".xSafetyState);
END_REGION

REGION Network 6: Strat up warning
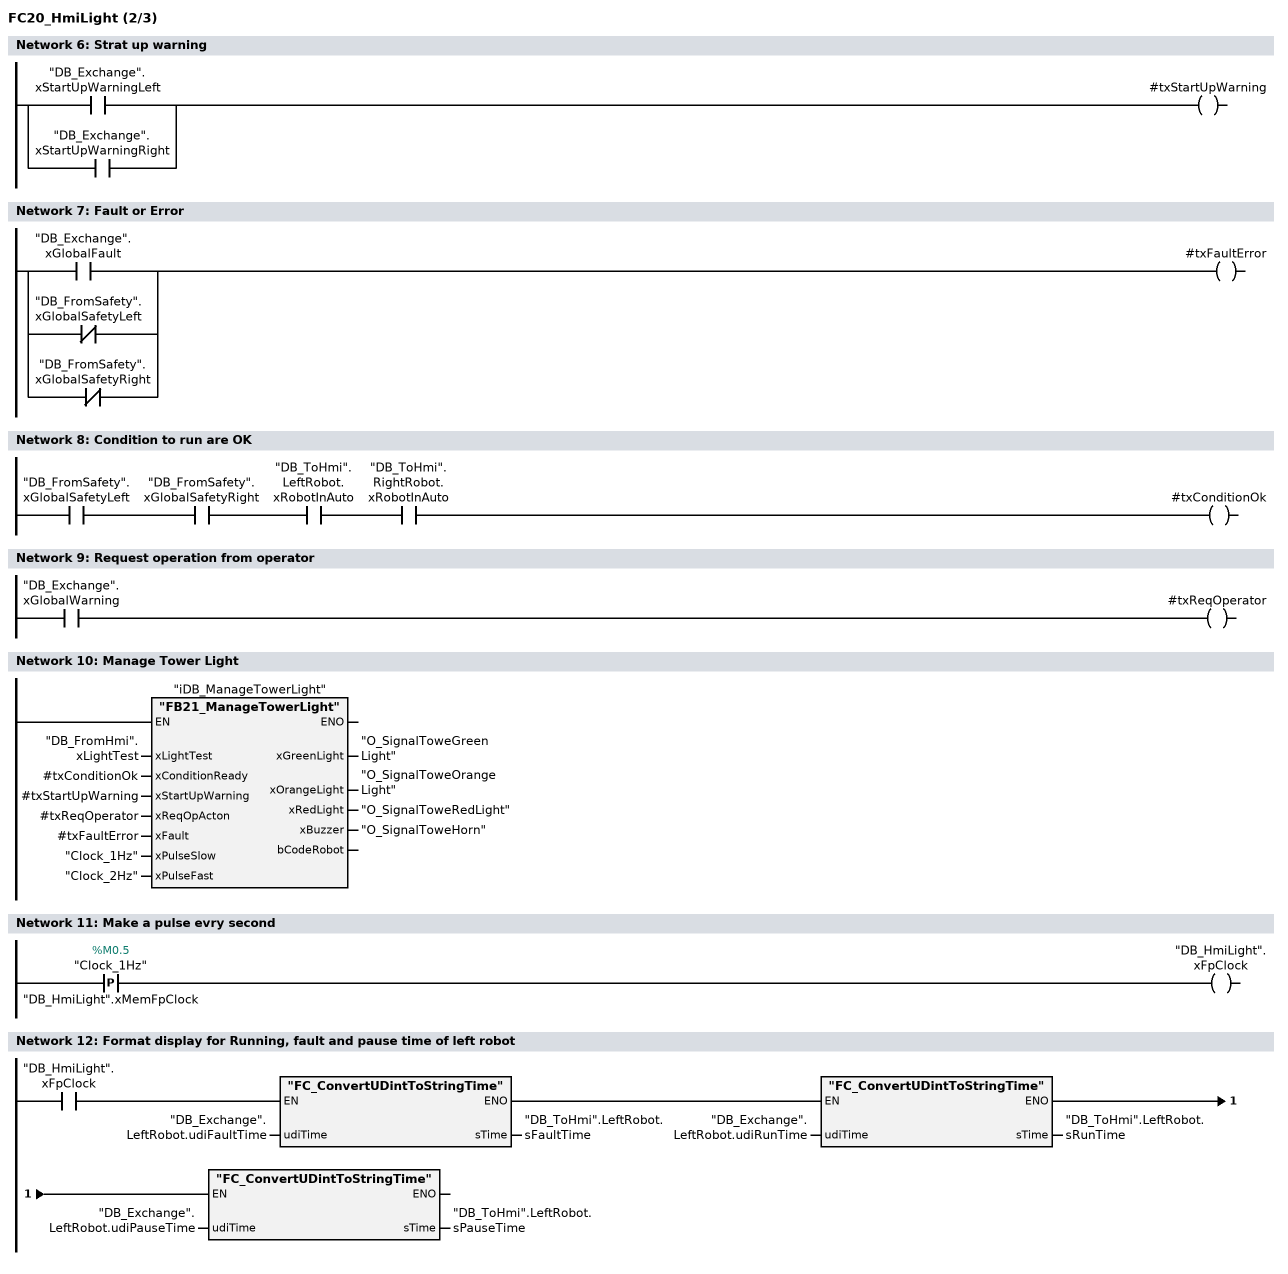
   RUNG wire#powerrail
      Contact( "DB_Exchange".xStartUpWarningLeft )
      wire#w1
      Coil( #txStartUpWarning )
   END_RUNG
   RUNG wire#powerrail
      Contact( "DB_Exchange".xStartUpWarningRight )
   END_RUNG wire#w1
   // the same network as SCL:
   #txStartUpWarning := "DB_Exchange".xStartUpWarningLeft OR "DB_Exchange".xStartUpWarningRight;
END_REGION

REGION Network 7: Fault or Error
   RUNG wire#powerrail
      Contact( "DB_Exchange".xGlobalFault )
      wire#w1
      Coil( #txFaultError )
   END_RUNG
   RUNG wire#powerrail
      I_Contact( "DB_FromSafety".xGlobalSafetyLeft )
   END_RUNG wire#w1
   RUNG wire#powerrail
      I_Contact( "DB_FromSafety".xGlobalSafetyRight )
   END_RUNG wire#w1
   // the same network as SCL:
   #txFaultError := "DB_Exchange".xGlobalFault OR NOT "DB_FromSafety".xGlobalSafetyLeft OR NOT "DB_FromSafety".xGlobalSafetyRight;
END_REGION

REGION Network 8: Condition to run are OK
   RUNG wire#powerrail
      Contact( "DB_FromSafety".xGlobalSafetyLeft )
      Contact( "DB_FromSafety".xGlobalSafetyRight )
      Contact( "DB_ToHmi".LeftRobot.xRobotInAuto )
      Contact( "DB_ToHmi".RightRobot.xRobotInAuto )
      Coil( #txConditionOk )
   END_RUNG
   // the same network as SCL:
   #txConditionOk := "DB_FromSafety".xGlobalSafetyLeft AND "DB_FromSafety".xGlobalSafetyRight AND "DB_ToHmi".LeftRobot.xRobotInAuto AND "DB_ToHmi".RightRobot.xRobotInAuto;
END_REGION

REGION Network 9: Request operation from operator
   RUNG wire#powerrail
      Contact( "DB_Exchange".xGlobalWarning )
      Coil( #txReqOperator )
   END_RUNG
   // the same network as SCL:
   #txReqOperator := "DB_Exchange".xGlobalWarning;
END_REGION

REGION Network 10: Manage Tower Light
   RUNG wire#powerrail
      "iDB_ManageTowerLight"(xLightTest := "DB_FromHmi".xLightTest, xConditionReady := #txConditionOk, xStartUpWarning := #txStartUpWarning, xReqOpActon := #txReqOperator, xFault := #txFaultError, xPulseSlow := "Clock_1Hz", xPulseFast := "Clock_2Hz", xGreenLight => "O_SignalToweGreenLight", xOrangeLight => "O_SignalToweOrangeLight", xRedLight => "O_SignalToweRedLight", xBuzzer => "O_SignalToweHorn", bCodeRobot =>)
   END_RUNG
   // the same network as SCL:
   "iDB_ManageTowerLight"(xLightTest := "DB_FromHmi".xLightTest,   // "FB21_ManageTowerLight"
                          xConditionReady := #txConditionOk,
                          xStartUpWarning := #txStartUpWarning,
                          xReqOpActon := #txReqOperator,
                          xFault := #txFaultError,
                          xPulseSlow := "Clock_1Hz",
                          xPulseFast := "Clock_2Hz",
                          xGreenLight => "O_SignalToweGreenLight",
                          xOrangeLight => "O_SignalToweOrangeLight",
                          xRedLight => "O_SignalToweRedLight",
                          xBuzzer => "O_SignalToweHorn");
END_REGION

REGION Network 11: Make a pulse evry second
   RUNG wire#powerrail
      P_Contact(operand := "Clock_1Hz", bit := "DB_HmiLight".xMemFpClock)
      Coil( "DB_HmiLight".xFpClock )
   END_RUNG
   // the same network as SCL:
   #_w1 := "Clock_1Hz" AND NOT "DB_HmiLight".xMemFpClock;   // rising edge of "Clock_1Hz"
   "DB_HmiLight".xMemFpClock := "Clock_1Hz";
   "DB_HmiLight".xFpClock := #_w1;
END_REGION

REGION Network 12: Format display for Running, fault and pause time of left robot
   RUNG wire#powerrail
      Contact( "DB_HmiLight".xFpClock )
      "FC_ConvertUDintToStringTime"(udiTime := "DB_Exchange".LeftRobot.udiFaultTime, sTime => "DB_ToHmi".LeftRobot.sFaultTime)
      "FC_ConvertUDintToStringTime"(udiTime := "DB_Exchange".LeftRobot.udiRunTime, sTime => "DB_ToHmi".LeftRobot.sRunTime)
      "FC_ConvertUDintToStringTime"(udiTime := "DB_Exchange".LeftRobot.udiPauseTime, sTime => "DB_ToHmi".LeftRobot.sPauseTime)
   END_RUNG
   // the same network as SCL:
   "FC_ConvertUDintToStringTime"(EN := "DB_HmiLight".xFpClock,
                           udiTime := "DB_Exchange".LeftRobot.udiFaultTime,
                           sTime => "DB_ToHmi".LeftRobot.sFaultTime,
                           ENO => #_w1);
   "FC_ConvertUDintToStringTime"(EN := #_w1,
                           udiTime := "DB_Exchange".LeftRobot.udiRunTime,
                           sTime => "DB_ToHmi".LeftRobot.sRunTime,
                           ENO => #_w2);
   IF #_w2 THEN
       "FC_ConvertUDintToStringTime"(udiTime := "DB_Exchange".LeftRobot.udiPauseTime,
                               sTime => "DB_ToHmi".LeftRobot.sPauseTime);
   END_IF;
END_REGION

REGION Network 13: Format display for Robot power on et robto drive on time of left robot
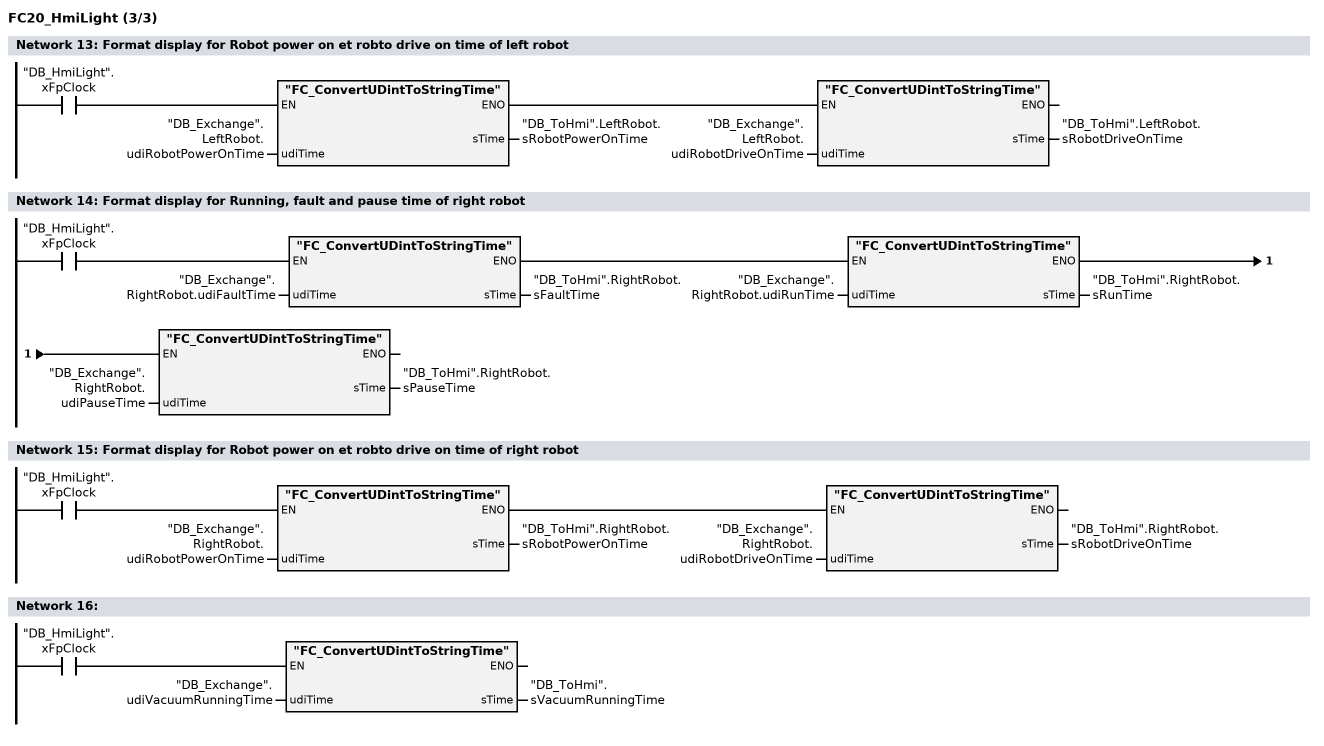
   RUNG wire#powerrail
      Contact( "DB_HmiLight".xFpClock )
      "FC_ConvertUDintToStringTime"(udiTime := "DB_Exchange".LeftRobot.udiRobotPowerOnTime, sTime => "DB_ToHmi".LeftRobot.sRobotPowerOnTime)
      "FC_ConvertUDintToStringTime"(udiTime := "DB_Exchange".LeftRobot.udiRobotDriveOnTime, sTime => "DB_ToHmi".LeftRobot.sRobotDriveOnTime)
   END_RUNG
   // the same network as SCL:
   "FC_ConvertUDintToStringTime"(EN := "DB_HmiLight".xFpClock,
                           udiTime := "DB_Exchange".LeftRobot.udiRobotPowerOnTime,
                           sTime => "DB_ToHmi".LeftRobot.sRobotPowerOnTime,
                           ENO => #_w1);
   IF #_w1 THEN
       "FC_ConvertUDintToStringTime"(udiTime := "DB_Exchange".LeftRobot.udiRobotDriveOnTime,
                               sTime => "DB_ToHmi".LeftRobot.sRobotDriveOnTime);
   END_IF;
END_REGION

REGION Network 14: Format display for Running, fault and pause time of right robot
   RUNG wire#powerrail
      Contact( "DB_HmiLight".xFpClock )
      "FC_ConvertUDintToStringTime"(udiTime := "DB_Exchange".RightRobot.udiFaultTime, sTime => "DB_ToHmi".RightRobot.sFaultTime)
      "FC_ConvertUDintToStringTime"(udiTime := "DB_Exchange".RightRobot.udiRunTime, sTime => "DB_ToHmi".RightRobot.sRunTime)
      "FC_ConvertUDintToStringTime"(udiTime := "DB_Exchange".RightRobot.udiPauseTime, sTime => "DB_ToHmi".RightRobot.sPauseTime)
   END_RUNG
   // the same network as SCL:
   "FC_ConvertUDintToStringTime"(EN := "DB_HmiLight".xFpClock,
                           udiTime := "DB_Exchange".RightRobot.udiFaultTime,
                           sTime => "DB_ToHmi".RightRobot.sFaultTime,
                           ENO => #_w1);
   "FC_ConvertUDintToStringTime"(EN := #_w1,
                           udiTime := "DB_Exchange".RightRobot.udiRunTime,
                           sTime => "DB_ToHmi".RightRobot.sRunTime,
                           ENO => #_w2);
   IF #_w2 THEN
       "FC_ConvertUDintToStringTime"(udiTime := "DB_Exchange".RightRobot.udiPauseTime,
                               sTime => "DB_ToHmi".RightRobot.sPauseTime);
   END_IF;
END_REGION

REGION Network 15: Format display for Robot power on et robto drive on time of right robot
   RUNG wire#powerrail
      Contact( "DB_HmiLight".xFpClock )
      "FC_ConvertUDintToStringTime"(udiTime := "DB_Exchange".RightRobot.udiRobotPowerOnTime, sTime => "DB_ToHmi".RightRobot.sRobotPowerOnTime)
      "FC_ConvertUDintToStringTime"(udiTime := "DB_Exchange".RightRobot.udiRobotDriveOnTime, sTime => "DB_ToHmi".RightRobot.sRobotDriveOnTime)
   END_RUNG
   // the same network as SCL:
   "FC_ConvertUDintToStringTime"(EN := "DB_HmiLight".xFpClock,
                           udiTime := "DB_Exchange".RightRobot.udiRobotPowerOnTime,
                           sTime => "DB_ToHmi".RightRobot.sRobotPowerOnTime,
                           ENO => #_w1);
   IF #_w1 THEN
       "FC_ConvertUDintToStringTime"(udiTime := "DB_Exchange".RightRobot.udiRobotDriveOnTime,
                               sTime => "DB_ToHmi".RightRobot.sRobotDriveOnTime);
   END_IF;
END_REGION

REGION Network 16
   RUNG wire#powerrail
      Contact( "DB_HmiLight".xFpClock )
      "FC_ConvertUDintToStringTime"(udiTime := "DB_Exchange".udiVacuumRunningTime, sTime => "DB_ToHmi".sVacuumRunningTime)
   END_RUNG
   // the same network as SCL:
   IF "DB_HmiLight".xFpClock THEN
       "FC_ConvertUDintToStringTime"(udiTime := "DB_Exchange".udiVacuumRunningTime,
                               sTime => "DB_ToHmi".sVacuumRunningTime);
   END_IF;
END_REGION

REGION Network 17 (SCL): Copy status to HMI
   "DB_ToHmi".xAccessDoor := "DB_FromSafety".DoorAcces.State;
   "DB_ToHmi".xCaptiveKey := "DB_FromSafety".CaptiveKeyInLock.State;
   "DB_ToHmi".xLightBeam := "DB_FromSafety".PedestrialDoorAcces.State;
   "DB_ToHmi".xCbsGate := "DB_FromSafety".GateAccesCBS.State;
END_REGION
END_FUNCTION

FUNCTION_BLOCK "FB20_ManageState"   // FB20, LAD
{ S7_Optimized_Access := 'TRUE' }
// stored: AutoNumber false, IsIECCheckEnabled true, MemoryReserve 100, SetENOAutomatically false
   VAR_INPUT
      xGlobalSafety { ExternalAccessible := 'False'; ExternalVisible := 'False'; ExternalWritable := 'False'} : Bool;
      xGlobalFault { ExternalAccessible := 'False'; ExternalVisible := 'False'; ExternalWritable := 'False'} : Bool;
      xInformation { ExternalAccessible := 'False'; ExternalVisible := 'False'; ExternalWritable := 'False'} : Bool;
   END_VAR
   VAR_OUTPUT
      nGlobalState { ExternalAccessible := 'False'; ExternalVisible := 'False'; ExternalWritable := 'False'} : Int;
      xSafetyState { ExternalAccessible := 'False'; ExternalVisible := 'False'; ExternalWritable := 'False'} : Bool;
   END_VAR
BEGIN

REGION Network 1: Safety fault
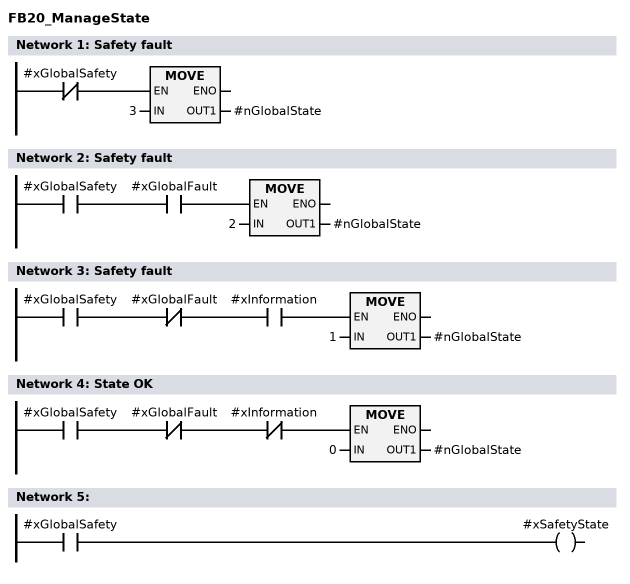
   RUNG wire#powerrail
      I_Contact( #xGlobalSafety )
      Move(in := 3, out1 => #nGlobalState)
   END_RUNG
   // the same network as SCL:
   IF NOT #xGlobalSafety THEN #nGlobalState := 3; END_IF;
END_REGION

REGION Network 2: Safety fault
   RUNG wire#powerrail
      Contact( #xGlobalSafety )
      Contact( #xGlobalFault )
      Move(in := 2, out1 => #nGlobalState)
   END_RUNG
   // the same network as SCL:
   IF #xGlobalSafety AND #xGlobalFault THEN #nGlobalState := 2; END_IF;
END_REGION

REGION Network 3: Safety fault
   RUNG wire#powerrail
      Contact( #xGlobalSafety )
      I_Contact( #xGlobalFault )
      Contact( #xInformation )
      Move(in := 1, out1 => #nGlobalState)
   END_RUNG
   // the same network as SCL:
   IF #xGlobalSafety AND NOT #xGlobalFault AND #xInformation THEN #nGlobalState := 1; END_IF;
END_REGION

REGION Network 4: State OK
   RUNG wire#powerrail
      Contact( #xGlobalSafety )
      I_Contact( #xGlobalFault )
      I_Contact( #xInformation )
      Move(in := 0, out1 => #nGlobalState)
   END_RUNG
   // the same network as SCL:
   IF #xGlobalSafety AND NOT #xGlobalFault AND NOT #xInformation THEN #nGlobalState := 0; END_IF;
END_REGION

REGION Network 5
   RUNG wire#powerrail
      Contact( #xGlobalSafety )
      Coil( #xSafetyState )
   END_RUNG
   // the same network as SCL:
   #xSafetyState := #xGlobalSafety;
END_REGION
END_FUNCTION_BLOCK

FUNCTION_BLOCK "FB21_ManageTowerLight"   // FB21, LAD
{ S7_Optimized_Access := 'TRUE' }
// stored: AutoNumber false, IsIECCheckEnabled true, MemoryReserve 100, SetENOAutomatically false
   VAR_INPUT
      xLightTest { ExternalAccessible := 'False'; ExternalVisible := 'False'; ExternalWritable := 'False'} : Bool;   // Light test
      xConditionReady { ExternalAccessible := 'False'; ExternalVisible := 'False'; ExternalWritable := 'False'} : Bool;   // All condition are Ok
      xStartUpWarning { ExternalAccessible := 'False'; ExternalVisible := 'False'; ExternalWritable := 'False'} : Bool;   // Warning before start
      xReqOpActon { ExternalAccessible := 'False'; ExternalVisible := 'False'; ExternalWritable := 'False'} : Bool;   // Requered Operator action
      xFault { ExternalAccessible := 'False'; ExternalVisible := 'False'; ExternalWritable := 'False'} : Bool;   // Fault or safety
      xPulseSlow { ExternalAccessible := 'False'; ExternalVisible := 'False'; ExternalWritable := 'False'} : Bool;   // Pulse slow
      xPulseFast { ExternalAccessible := 'False'; ExternalVisible := 'False'; ExternalWritable := 'False'} : Bool;   // Pulse fast
   END_VAR
   VAR_OUTPUT
      xGreenLight { ExternalAccessible := 'False'; ExternalVisible := 'False'; ExternalWritable := 'False'} : Bool;   // Tower Green Light
      xOrangeLight { ExternalAccessible := 'False'; ExternalVisible := 'False'; ExternalWritable := 'False'} : Bool;   // Tower Orrange Light
      xRedLight { ExternalAccessible := 'False'; ExternalVisible := 'False'; ExternalWritable := 'False'} : Bool;   // Tower Red Light
      xBuzzer { ExternalAccessible := 'False'; ExternalVisible := 'False'; ExternalWritable := 'False'} : Bool;   // Tower Buzzer
      bCodeRobot { ExternalAccessible := 'False'; ExternalVisible := 'False'; ExternalWritable := 'False'} : Byte;   // Code state for robot
   END_VAR
   VAR
      miDB_TpNewFault { ExternalAccessible := 'False'; ExternalVisible := 'False'; ExternalWritable := 'False'; S7_SetPoint := 'True'} : TP_TIME;
   END_VAR
   VAR_TEMP   // added for the SCL form of the ladder/FBD networks
      _w1 : Bool;
   END_VAR
BEGIN

REGION Network 1: Reset byte code Robot
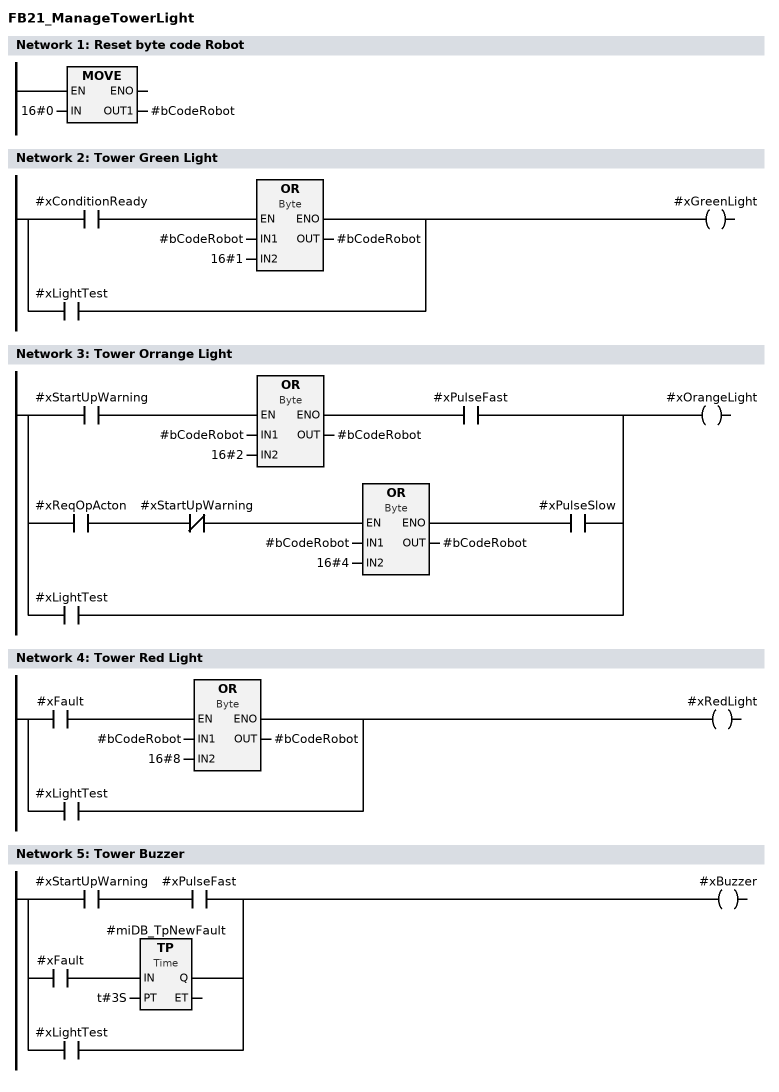
   RUNG wire#powerrail
      Move(in := 16#0, out1 => #bCodeRobot)
   END_RUNG
   // the same network as SCL:
   #bCodeRobot := 16#0;
END_REGION

REGION Network 2: Tower Green Light
   IF #xConditionReady THEN #bCodeRobot := #bCodeRobot OR 16#1; END_IF;
   #xGreenLight := #xConditionReady OR #xLightTest;
END_REGION

REGION Network 3: Tower Orrange Light
   IF #xStartUpWarning THEN #bCodeRobot := #bCodeRobot OR 16#2; END_IF;
   #_w1 := #xReqOpActon AND NOT #xStartUpWarning;
   IF #_w1 THEN #bCodeRobot := #bCodeRobot OR 16#4; END_IF;
   #xOrangeLight := (#xStartUpWarning AND #xPulseFast) OR (#_w1 AND #xPulseSlow) OR #xLightTest;
END_REGION

REGION Network 4: Tower Red Light
   IF #xFault THEN #bCodeRobot := #bCodeRobot OR 16#8; END_IF;
   #xRedLight := #xFault OR #xLightTest;
END_REGION

REGION Network 5: Tower Buzzer
   RUNG wire#powerrail
      Contact( #xStartUpWarning )
      Contact( #xPulseFast )
      wire#w1
      Coil( #xBuzzer )
   END_RUNG
   RUNG wire#powerrail
      Contact( #xFault )
      { S7_Templates := "time_type := Time" } #miDB_TpNewFault.TP(pt := t#3S, et =>)
   END_RUNG wire#w1
   RUNG wire#powerrail
      Contact( #xLightTest )
   END_RUNG wire#w1
   // the same network as SCL:
   #miDB_TpNewFault(IN := #xFault, PT := t#3S);   // TP
   #xBuzzer := (#xStartUpWarning AND #xPulseFast) OR #miDB_TpNewFault.Q OR #xLightTest;
END_REGION
END_FUNCTION_BLOCK

FUNCTION "FC_ConvertUDintToStringTime" : Void
{ S7_Optimized_Access := 'TRUE' }
VERSION : 0.1
   VAR_INPUT 
      udiTime : UDInt;
   END_VAR

   VAR_OUTPUT 
      sTime : String;
   END_VAR

   VAR_TEMP 
      tudiTemp : UDInt;
      tudiTempHour : UDInt;
      tudiTempMinute : UDInt;
      tudiTempSeconde : UDInt;
      tsTmp : String;
      tsHour : String;
      tsMinute : String;
      tsSecond : String;
   END_VAR

   VAR CONSTANT 
      cSecondHour : UDInt := 3600;
      cSecondMinute : UDInt := 60;
   END_VAR


BEGIN
	// Reset Time
	#sTime := '';
	
	// Calcul hour
	IF #udiTime >= #cSecondHour THEN
	  #tudiTempHour := #udiTime / #cSecondHour;
	  #tsTmp := DELETE(IN := UDINT_TO_STRING(#tudiTempHour), L := 1, P := 1);
	  #tsHour := CONCAT_STRING(IN1 := #tsTmp, IN2 := 'h ');
	  #tudiTemp := (#udiTime - (#tudiTempHour * #cSecondHour));
	ELSE
	  #tsHour := '0h ';
	  #tudiTemp := #udiTime;
	END_IF;
	
	// Calcul Minutes
	#tudiTempMinute := #tudiTemp / #cSecondMinute;
	#tsTmp := DELETE(IN := UDINT_TO_STRING(#tudiTempMinute), L := 1, P := 1);
	IF #tudiTempMinute = 0 THEN
	  #tsMinute := '00';
	ELSIF #tudiTempMinute < 10 THEN
	  #tsMinute := CONCAT(IN1 := '0', IN2 := #tsTmp);
	ELSE
	  #tsMinute := #tsTmp;
	END_IF;
	#tsMinute := CONCAT_STRING(IN1 := #tsMinute, IN2 := 'm ');
	#tudiTemp := (#tudiTemp - (#tudiTempMinute * #cSecondMinute));
	
	// Calcul Seconds
	#tudiTempSeconde := #tudiTemp;
	#tsTmp := DELETE(IN := UDINT_TO_STRING(#tudiTempSeconde), L := 1, P := 1);
	IF #tudiTempSeconde = 0 THEN
	  #tsSecond := '00';
	ELSIF #tudiTempSeconde < 10 THEN
	  #tsSecond := CONCAT(IN1 := '0', IN2 := #tsTmp);
	ELSE
	  #tsSecond := #tsTmp;
	END_IF;
	#tsSecond := CONCAT_STRING(IN1 := #tsSecond, IN2 := 's');
	
	#sTime := CONCAT(IN1 := #tsHour, IN2 := #tsMinute);
	#sTime := CONCAT(IN1 := #sTime, IN2 := #tsSecond);
	
	
END_FUNCTION

FUNCTION "FC30_DoorAcces" : Void   // FC30, LAD
{ S7_Optimized_Access := 'TRUE' }
// stored: AutoNumber false, IsIECCheckEnabled true, SetENOAutomatically false
   VAR_TEMP
      xt_RobotStopped : Bool;
      xt_Robot1Stopped : Bool;
      xt_Robot2Stopped : Bool;
   END_VAR
BEGIN

REGION Network 1: Robot 1 is stopped
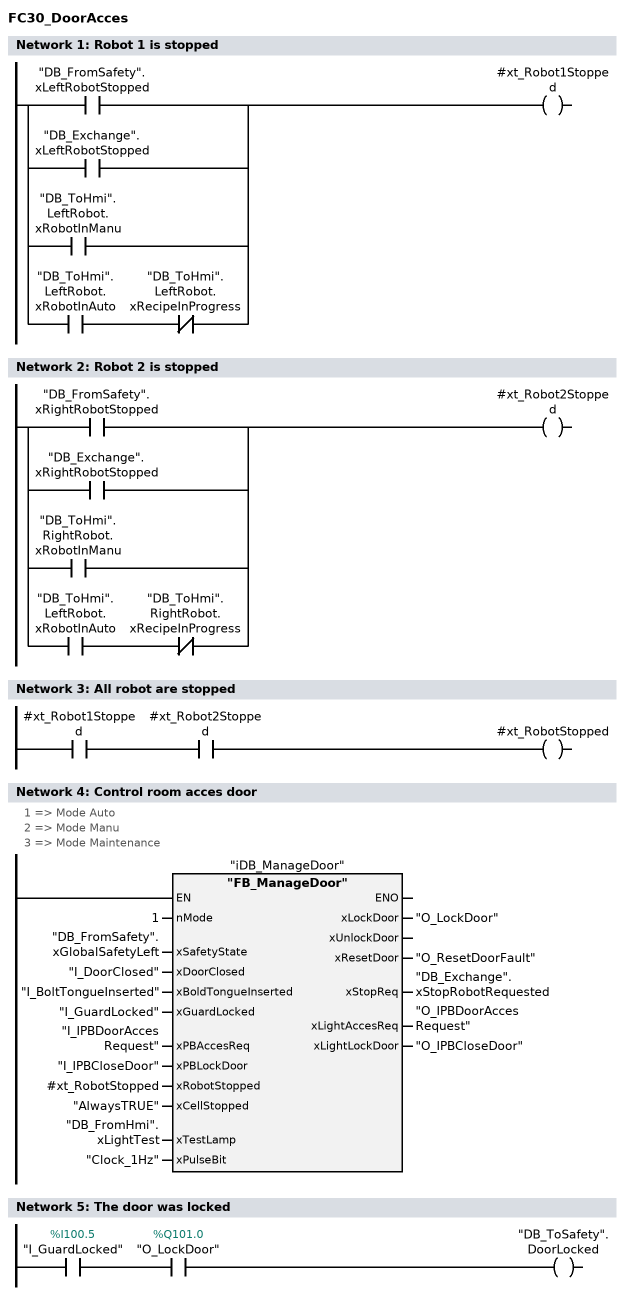
   RUNG wire#powerrail
      Contact( "DB_FromSafety".xLeftRobotStopped )
      wire#w1
      Coil( #xt_Robot1Stopped )
   END_RUNG
   RUNG wire#powerrail
      Contact( "DB_Exchange".xLeftRobotStopped )
   END_RUNG wire#w1
   RUNG wire#powerrail
      Contact( "DB_ToHmi".LeftRobot.xRobotInManu )
   END_RUNG wire#w1
   RUNG wire#powerrail
      Contact( "DB_ToHmi".LeftRobot.xRobotInAuto )
      I_Contact( "DB_ToHmi".LeftRobot.xRecipeInProgress )
   END_RUNG wire#w1
   // the same network as SCL:
   #xt_Robot1Stopped := "DB_FromSafety".xLeftRobotStopped OR "DB_Exchange".xLeftRobotStopped OR "DB_ToHmi".LeftRobot.xRobotInManu OR ("DB_ToHmi".LeftRobot.xRobotInAuto AND NOT "DB_ToHmi".LeftRobot.xRecipeInProgress);
END_REGION

REGION Network 2: Robot 2 is stopped
   RUNG wire#powerrail
      Contact( "DB_FromSafety".xRightRobotStopped )
      wire#w1
      Coil( #xt_Robot2Stopped )
   END_RUNG
   RUNG wire#powerrail
      Contact( "DB_Exchange".xRightRobotStopped )
   END_RUNG wire#w1
   RUNG wire#powerrail
      Contact( "DB_ToHmi".RightRobot.xRobotInManu )
   END_RUNG wire#w1
   RUNG wire#powerrail
      Contact( "DB_ToHmi".LeftRobot.xRobotInAuto )
      I_Contact( "DB_ToHmi".RightRobot.xRecipeInProgress )
   END_RUNG wire#w1
   // the same network as SCL:
   #xt_Robot2Stopped := "DB_FromSafety".xRightRobotStopped OR "DB_Exchange".xRightRobotStopped OR "DB_ToHmi".RightRobot.xRobotInManu OR ("DB_ToHmi".LeftRobot.xRobotInAuto AND NOT "DB_ToHmi".RightRobot.xRecipeInProgress);
END_REGION

REGION Network 3: All robot are stopped
   RUNG wire#powerrail
      Contact( #xt_Robot1Stopped )
      Contact( #xt_Robot2Stopped )
      Coil( #xt_RobotStopped )
   END_RUNG
   // the same network as SCL:
   #xt_RobotStopped := #xt_Robot1Stopped AND #xt_Robot2Stopped;
END_REGION

REGION Network 4: Control room acces door
   // 1 => Mode Auto
   // 2 => Mode Manu
   // 3 => Mode Maintenance
   RUNG wire#powerrail
      "iDB_ManageDoor"(nMode := 1, xSafetyState := "DB_FromSafety".xGlobalSafetyLeft, xDoorClosed := "I_DoorClosed", xBoldTongueInserted := "I_BoltTongueInserted", xGuardLocked := "I_GuardLocked", xPBAccesReq := "I_IPBDoorAccesRequest", xPBLockDoor := "I_IPBCloseDoor", xRobotStopped := #xt_RobotStopped, xCellStopped := "AlwaysTRUE", xTestLamp := "DB_FromHmi".xLightTest, xPulseBit := "Clock_1Hz", xLockDoor => "O_LockDoor", xUnlockDoor =>, xResetDoor => "O_ResetDoorFault", xStopReq => "DB_Exchange".xStopRobotRequested, xLightAccesReq => "O_IPBDoorAccesRequest", xLightLockDoor => "O_IPBCloseDoor")
   END_RUNG
   // the same network as SCL:
   "iDB_ManageDoor"(nMode := 1,   // "FB_ManageDoor"
                    xSafetyState := "DB_FromSafety".xGlobalSafetyLeft,
                    xDoorClosed := "I_DoorClosed",
                    xBoldTongueInserted := "I_BoltTongueInserted",
                    xGuardLocked := "I_GuardLocked",
                    xPBAccesReq := "I_IPBDoorAccesRequest",
                    xPBLockDoor := "I_IPBCloseDoor",
                    xRobotStopped := #xt_RobotStopped,
                    xCellStopped := "AlwaysTRUE",
                    xTestLamp := "DB_FromHmi".xLightTest,
                    xPulseBit := "Clock_1Hz",
                    xLockDoor => "O_LockDoor",
                    xResetDoor => "O_ResetDoorFault",
                    xStopReq => "DB_Exchange".xStopRobotRequested,
                    xLightAccesReq => "O_IPBDoorAccesRequest",
                    xLightLockDoor => "O_IPBCloseDoor");
END_REGION

REGION Network 5: The door was locked
   RUNG wire#powerrail
      Contact( "I_GuardLocked" )
      Contact( "O_LockDoor" )
      Coil( "DB_ToSafety".DoorLocked )
   END_RUNG
   // the same network as SCL:
   "DB_ToSafety".DoorLocked := "I_GuardLocked" AND "O_LockDoor";
END_REGION
END_FUNCTION

FUNCTION_BLOCK "FB_ManageDoor"   // FB1010, LAD
{ S7_Optimized_Access := 'TRUE' }
// stored: AutoNumber false, MemoryReserve 100, SetENOAutomatically false
   VAR_INPUT
      nMode { ExternalAccessible := 'False'; ExternalVisible := 'False'; ExternalWritable := 'False'} : Int;
      xSafetyState { ExternalAccessible := 'False'; ExternalVisible := 'False'; ExternalWritable := 'False'} : Bool;
      xDoorClosed { ExternalAccessible := 'False'; ExternalVisible := 'False'; ExternalWritable := 'False'} : Bool;   // ON when the door is closed
      xBoldTongueInserted { ExternalAccessible := 'False'; ExternalVisible := 'False'; ExternalWritable := 'False'} : Bool;   // Bolt tongue inserted into the evaluation module
      xGuardLocked { ExternalAccessible := 'False'; ExternalVisible := 'False'; ExternalWritable := 'False'} : Bool;   // Guard locking solenoid in locked position
      xPBAccesReq { ExternalAccessible := 'False'; ExternalVisible := 'False'; ExternalWritable := 'False'} : Bool;
      xPBLockDoor { ExternalAccessible := 'False'; ExternalVisible := 'False'; ExternalWritable := 'False'} : Bool;
      xRobotStopped { ExternalAccessible := 'False'; ExternalVisible := 'False'; ExternalWritable := 'False'} : Bool;
      xCellStopped { ExternalAccessible := 'False'; ExternalVisible := 'False'; ExternalWritable := 'False'} : Bool;
      xTestLamp { ExternalAccessible := 'False'; ExternalVisible := 'False'; ExternalWritable := 'False'} : Bool;
      xPulseBit { ExternalAccessible := 'False'; ExternalVisible := 'False'; ExternalWritable := 'False'} : Bool;
   END_VAR
   VAR_OUTPUT
      xLockDoor { ExternalAccessible := 'False'; ExternalVisible := 'False'; ExternalWritable := 'False'} : Bool;
      xUnlockDoor { ExternalAccessible := 'False'; ExternalVisible := 'False'; ExternalWritable := 'False'} : Bool;
      xResetDoor { ExternalAccessible := 'False'; ExternalVisible := 'False'; ExternalWritable := 'False'} : Bool;
      xStopReq { ExternalAccessible := 'False'; ExternalVisible := 'False'; ExternalWritable := 'False'} : Bool;
      xLightAccesReq { ExternalAccessible := 'False'; ExternalVisible := 'False'; ExternalWritable := 'False'} : Bool;
      xLightLockDoor { ExternalAccessible := 'False'; ExternalVisible := 'False'; ExternalWritable := 'False'} : Bool;
   END_VAR
   VAR
      sFPAccesReq { ExternalAccessible := 'False'; ExternalVisible := 'False'; ExternalWritable := 'False'} : Bool;
      sxAccesRequested { ExternalAccessible := 'False'; ExternalVisible := 'False'; ExternalWritable := 'False'} : Bool;
      sxAccesAllowed { ExternalAccessible := 'False'; ExternalVisible := 'False'; ExternalWritable := 'False'} : Bool;
   END_VAR
   VAR_TEMP
      tAccesReq : Bool;
   END_VAR
   VAR CONSTANT
      ModeAuto : Int := 1;
      ModeManu : Int := 2;
      ModeMaintenance : Int := 3;
   END_VAR
   VAR_TEMP   // added for the SCL form of the ladder/FBD networks
      _w1 : Bool;
      _w2 : Bool;
   END_VAR
BEGIN

REGION Network 1: Set and Reset internal acces request
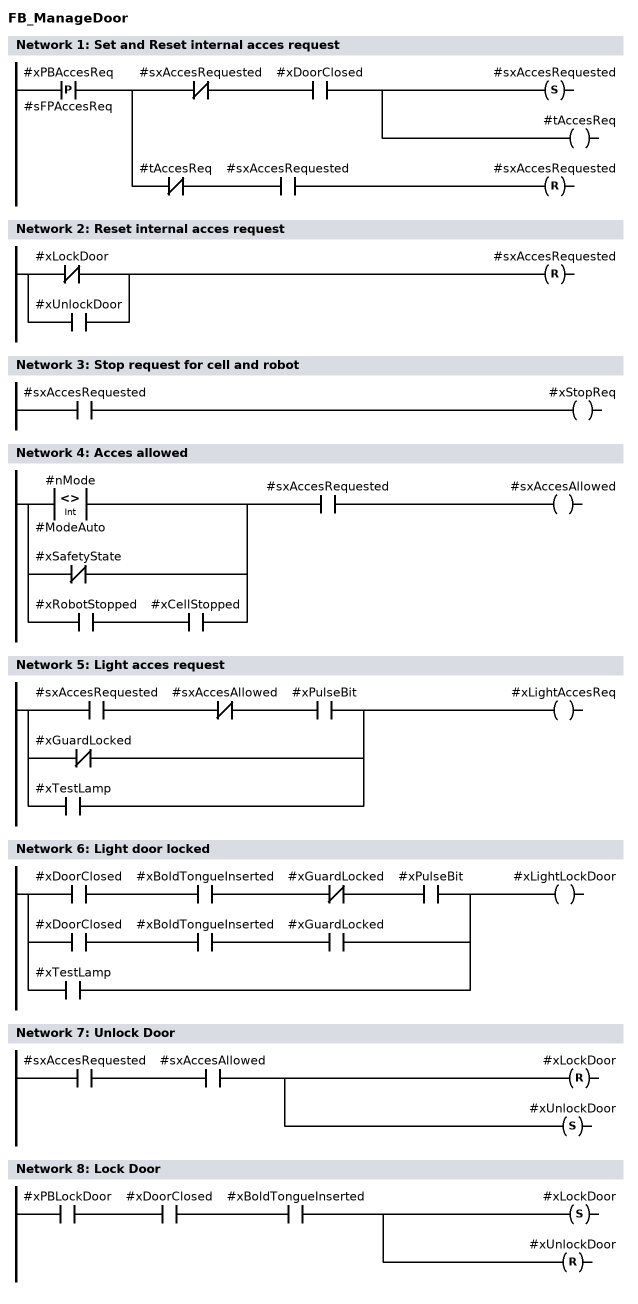
   RUNG wire#powerrail
      P_Contact(operand := #xPBAccesReq, bit := #sFPAccesReq)
      wire#w1
      I_Contact( #sxAccesRequested )
      Contact( #xDoorClosed )
      wire#w2
      S_Coil( #sxAccesRequested )
   END_RUNG
   RUNG wire#w2
      Coil( #tAccesReq )
   END_RUNG
   RUNG wire#w1
      I_Contact( #tAccesReq )
      Contact( #sxAccesRequested )
      R_Coil( #sxAccesRequested )
   END_RUNG
   // the same network as SCL:
   #_w1 := #xPBAccesReq AND NOT #sFPAccesReq;   // rising edge of #xPBAccesReq
   #sFPAccesReq := #xPBAccesReq;
   #_w2 := #_w1 AND NOT #sxAccesRequested AND #xDoorClosed;
   IF #_w2 THEN #sxAccesRequested := TRUE; END_IF;
   #tAccesReq := #_w2;
   IF #_w1 AND NOT #tAccesReq AND #sxAccesRequested THEN #sxAccesRequested := FALSE; END_IF;
END_REGION

REGION Network 2: Reset internal acces request
   RUNG wire#powerrail
      I_Contact( #xLockDoor )
      wire#w1
      R_Coil( #sxAccesRequested )
   END_RUNG
   RUNG wire#powerrail
      Contact( #xUnlockDoor )
   END_RUNG wire#w1
   // the same network as SCL:
   IF NOT #xLockDoor OR #xUnlockDoor THEN #sxAccesRequested := FALSE; END_IF;
END_REGION

REGION Network 3: Stop request for cell and robot
   RUNG wire#powerrail
      Contact( #sxAccesRequested )
      Coil( #xStopReq )
   END_RUNG
   // the same network as SCL:
   #xStopReq := #sxAccesRequested;
END_REGION

REGION Network 4: Acces allowed
   RUNG wire#powerrail
      { S7_Templates := "SrcType := Int" } NE_Contact(in1 := #nMode, in2 := #ModeAuto)
      wire#w1
      Contact( #sxAccesRequested )
      Coil( #sxAccesAllowed )
   END_RUNG
   RUNG wire#powerrail
      I_Contact( #xSafetyState )
   END_RUNG wire#w1
   RUNG wire#powerrail
      Contact( #xRobotStopped )
      Contact( #xCellStopped )
   END_RUNG wire#w1
   // the same network as SCL:
   #sxAccesAllowed := ((#nMode <> #ModeAuto) OR NOT #xSafetyState OR (#xRobotStopped AND #xCellStopped)) AND #sxAccesRequested;
END_REGION

REGION Network 5: Light acces request
   RUNG wire#powerrail
      Contact( #sxAccesRequested )
      I_Contact( #sxAccesAllowed )
      Contact( #xPulseBit )
      wire#w1
      Coil( #xLightAccesReq )
   END_RUNG
   RUNG wire#powerrail
      I_Contact( #xGuardLocked )
   END_RUNG wire#w1
   RUNG wire#powerrail
      Contact( #xTestLamp )
   END_RUNG wire#w1
   // the same network as SCL:
   #xLightAccesReq := (#sxAccesRequested AND NOT #sxAccesAllowed AND #xPulseBit) OR NOT #xGuardLocked OR #xTestLamp;
END_REGION

REGION Network 6: Light door locked
   RUNG wire#powerrail
      Contact( #xDoorClosed )
      Contact( #xBoldTongueInserted )
      I_Contact( #xGuardLocked )
      Contact( #xPulseBit )
      wire#w1
      Coil( #xLightLockDoor )
   END_RUNG
   RUNG wire#powerrail
      Contact( #xDoorClosed )
      Contact( #xBoldTongueInserted )
      Contact( #xGuardLocked )
   END_RUNG wire#w1
   RUNG wire#powerrail
      Contact( #xTestLamp )
   END_RUNG wire#w1
   // the same network as SCL:
   #xLightLockDoor := (#xDoorClosed AND #xBoldTongueInserted AND NOT #xGuardLocked AND #xPulseBit) OR (#xDoorClosed AND #xBoldTongueInserted AND #xGuardLocked) OR #xTestLamp;
END_REGION

REGION Network 7: Unlock Door
   RUNG wire#powerrail
      Contact( #sxAccesRequested )
      Contact( #sxAccesAllowed )
      wire#w1
      R_Coil( #xLockDoor )
   END_RUNG
   RUNG wire#w1
      S_Coil( #xUnlockDoor )
   END_RUNG
   // the same network as SCL:
   IF #sxAccesRequested AND #sxAccesAllowed THEN
       #xLockDoor := FALSE;
       #xUnlockDoor := TRUE;
   END_IF;
END_REGION

REGION Network 8: Lock Door
   RUNG wire#powerrail
      Contact( #xPBLockDoor )
      Contact( #xDoorClosed )
      Contact( #xBoldTongueInserted )
      wire#w1
      S_Coil( #xLockDoor )
   END_RUNG
   RUNG wire#w1
      R_Coil( #xUnlockDoor )
   END_RUNG
   // the same network as SCL:
   IF #xPBLockDoor AND #xDoorClosed AND #xBoldTongueInserted THEN
       #xLockDoor := TRUE;
       #xUnlockDoor := FALSE;
   END_IF;
END_REGION
END_FUNCTION_BLOCK

FUNCTION "FC40_CommSlave" : Void   // FC40, LAD
{ S7_Optimized_Access := 'TRUE' }
// stored: AutoNumber false, IsIECCheckEnabled true, SetENOAutomatically false
BEGIN

REGION Network 1: Manage communication with Left PLC
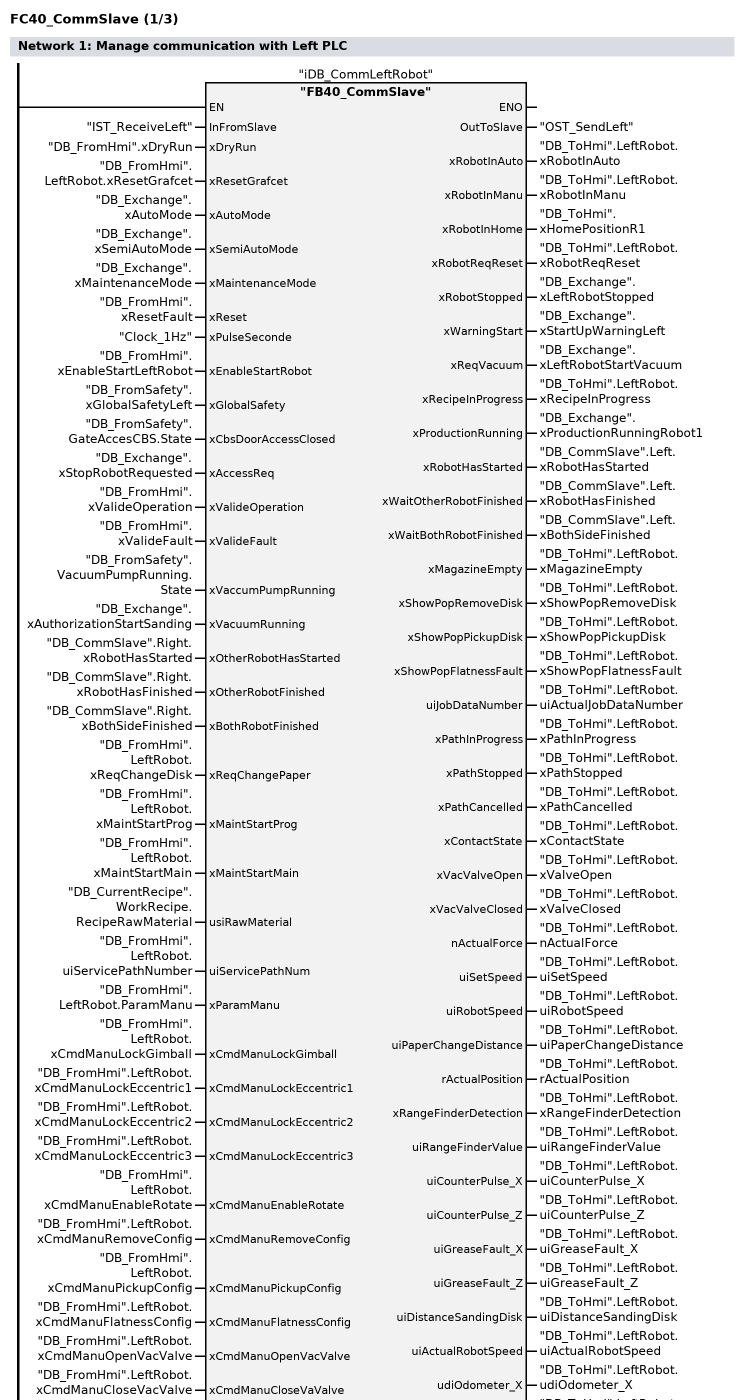
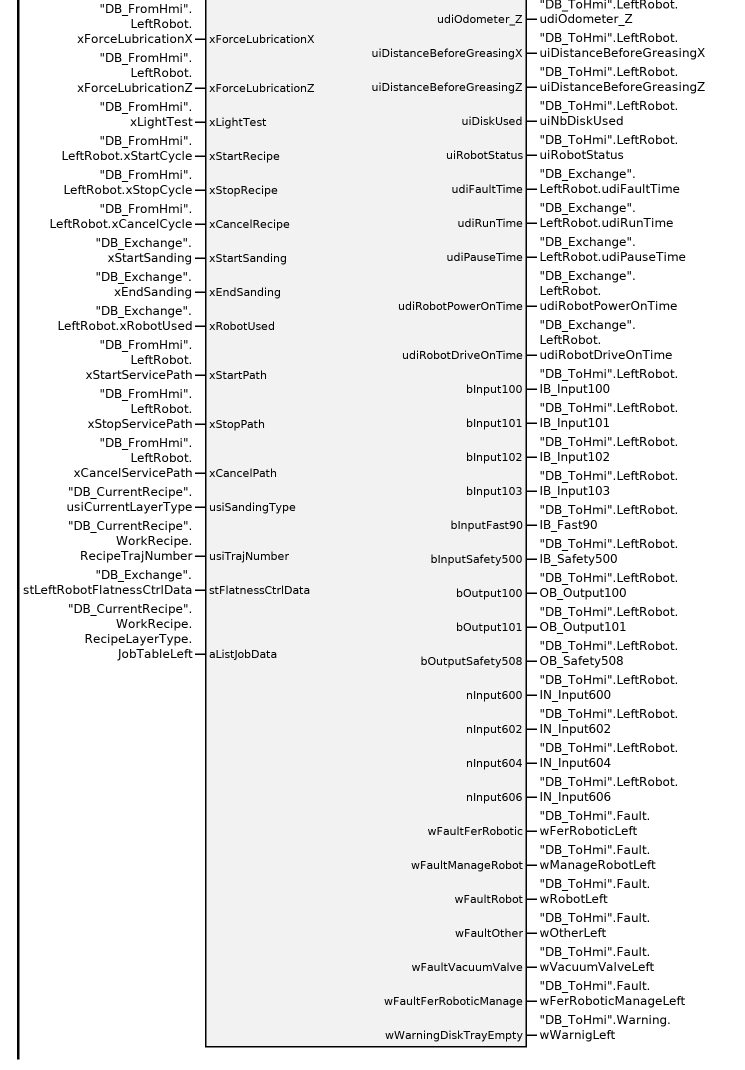
   RUNG wire#powerrail
      "iDB_CommLeftRobot"(InFromSlave := "IST_ReceiveLeft", xDryRun := "DB_FromHmi".xDryRun, xResetGrafcet := "DB_FromHmi".LeftRobot.xResetGrafcet, xAutoMode := "DB_Exchange".xAutoMode, xSemiAutoMode := "DB_Exchange".xSemiAutoMode, xMaintenanceMode := "DB_Exchange".xMaintenanceMode, xReset := "DB_FromHmi".xResetFault, xPulseSeconde := "Clock_1Hz", xEnableStartRobot := "DB_FromHmi".xEnableStartLeftRobot, xGlobalSafety := "DB_FromSafety".xGlobalSafetyLeft, xCbsDoorAccessClosed := "DB_FromSafety".GateAccesCBS.State, xAccessReq := "DB_Exchange".xStopRobotRequested, xValideOperation := "DB_FromHmi".xValideOperation, xValideFault := "DB_FromHmi".xValideFault, xVaccumPumpRunning := "DB_FromSafety".VacuumPumpRunning.State, xVacuumRunning := "DB_Exchange".xAuthorizationStartSanding, xOtherRobotHasStarted := "DB_CommSlave".Right.xRobotHasStarted, xOtherRobotFinished := "DB_CommSlave".Right.xRobotHasFinished, xBothRobotFinished := "DB_CommSlave".Right.xBothSideFinished, xReqChangePaper := "DB_FromHmi".LeftRobot.xReqChangeDisk, xMaintStartProg := "DB_FromHmi".LeftRobot.xMaintStartProg, xMaintStartMain := "DB_FromHmi".LeftRobot.xMaintStartMain, usiRawMaterial := "DB_CurrentRecipe".WorkRecipe.RecipeRawMaterial, uiServicePathNum := "DB_FromHmi".LeftRobot.uiServicePathNumber, xParamManu := "DB_FromHmi".LeftRobot.ParamManu, xCmdManuLockGimball := "DB_FromHmi".LeftRobot.xCmdManuLockGimball, xCmdManuLockEccentric1 := "DB_FromHmi".LeftRobot.xCmdManuLockEccentric1, xCmdManuLockEccentric2 := "DB_FromHmi".LeftRobot.xCmdManuLockEccentric2, xCmdManuLockEccentric3 := "DB_FromHmi".LeftRobot.xCmdManuLockEccentric3, xCmdManuEnableRotate := "DB_FromHmi".LeftRobot.xCmdManuEnableRotate, xCmdManuRemoveConfig := "DB_FromHmi".LeftRobot.xCmdManuRemoveConfig, xCmdManuPickupConfig := "DB_FromHmi".LeftRobot.xCmdManuPickupConfig, xCmdManuFlatnessConfig := "DB_FromHmi".LeftRobot.xCmdManuFlatnessConfig, xCmdManuOpenVacValve := "DB_FromHmi".LeftRobot.xCmdManuOpenVacValve, xCmdManuCloseVaValve := "DB_FromHmi".LeftRobot.xCmdManuCloseVacValve, xForceLubricationX := "DB_FromHmi".LeftRobot.xForceLubricationX, xForceLubricationZ := "DB_FromHmi".LeftRobot.xForceLubricationZ, xLightTest := "DB_FromHmi".xLightTest, xStartRecipe := "DB_FromHmi".LeftRobot.xStartCycle, xStopRecipe := "DB_FromHmi".LeftRobot.xStopCycle, xCancelRecipe := "DB_FromHmi".LeftRobot.xCancelCycle, xStartSanding := "DB_Exchange".xStartSanding, xEndSanding := "DB_Exchange".xEndSanding, xRobotUsed := "DB_Exchange".LeftRobot.xRobotUsed, xStartPath := "DB_FromHmi".LeftRobot.xStartServicePath, xStopPath := "DB_FromHmi".LeftRobot.xStopServicePath, xCancelPath := "DB_FromHmi".LeftRobot.xCancelServicePath, usiSandingType := "DB_CurrentRecipe".usiCurrentLayerType, usiTrajNumber := "DB_CurrentRecipe".WorkRecipe.RecipeTrajNumber, stFlatnessCtrlData := "DB_Exchange".stLeftRobotFlatnessCtrlData, aListJobData := "DB_CurrentRecipe".WorkRecipe.RecipeLayerType.JobTableLeft, OutToSlave => "OST_SendLeft", xRobotInAuto => "DB_ToHmi".LeftRobot.xRobotInAuto, xRobotInManu => "DB_ToHmi".LeftRobot.xRobotInManu, xRobotInHome => "DB_ToHmi".xHomePositionR1, xRobotReqReset => "DB_ToHmi".LeftRobot.xRobotReqReset, xRobotStopped => "DB_Exchange".xLeftRobotStopped, xWarningStart => "DB_Exchange".xStartUpWarningLeft, xReqVacuum => "DB_Exchange".xLeftRobotStartVacuum, xRecipeInProgress => "DB_ToHmi".LeftRobot.xRecipeInProgress, xProductionRunning => "DB_Exchange".xProductionRunningRobot1, xRobotHasStarted => "DB_CommSlave".Left.xRobotHasStarted, xWaitOtherRobotFinished => "DB_CommSlave".Left.xRobotHasFinished, xWaitBothRobotFinished => "DB_CommSlave".Left.xBothSideFinished, xMagazineEmpty => "DB_ToHmi".LeftRobot.xMagazineEmpty, xShowPopRemoveDisk => "DB_ToHmi".LeftRobot.xShowPopRemoveDisk, xShowPopPickupDisk => "DB_ToHmi".LeftRobot.xShowPopPickupDisk, xShowPopFlatnessFault => "DB_ToHmi".LeftRobot.xShowPopFlatnessFault, uiJobDataNumber => "DB_ToHmi".LeftRobot.uiActualJobDataNumber, xPathInProgress => "DB_ToHmi".LeftRobot.xPathInProgress, xPathStopped => "DB_ToHmi".LeftRobot.xPathStopped, xPathCancelled => "DB_ToHmi".LeftRobot.xPathCancelled, xContactState => "DB_ToHmi".LeftRobot.xContactState, xVacValveOpen => "DB_ToHmi".LeftRobot.xValveOpen, xVacValveClosed => "DB_ToHmi".LeftRobot.xValveClosed, nActualForce => "DB_ToHmi".LeftRobot.nActualForce, uiSetSpeed => "DB_ToHmi".LeftRobot.uiSetSpeed, uiRobotSpeed => "DB_ToHmi".LeftRobot.uiRobotSpeed, uiPaperChangeDistance => "DB_ToHmi".LeftRobot.uiPaperChangeDistance, rActualPosition => "DB_ToHmi".LeftRobot.rActualPosition, xRangeFinderDetection => "DB_ToHmi".LeftRobot.xRangeFinderDetection, uiRangeFinderValue => "DB_ToHmi".LeftRobot.uiRangeFinderValue, uiCounterPulse_X => "DB_ToHmi".LeftRobot.uiCounterPulse_X, uiCounterPulse_Z => "DB_ToHmi".LeftRobot.uiCounterPulse_Z, uiGreaseFault_X => "DB_ToHmi".LeftRobot.uiGreaseFault_X, uiGreaseFault_Z => "DB_ToHmi".LeftRobot.uiGreaseFault_Z, uiDistanceSandingDisk => "DB_ToHmi".LeftRobot.uiDistanceSandingDisk, uiActualRobotSpeed => "DB_ToHmi".LeftRobot.uiActualRobotSpeed, udiOdometer_X => "DB_ToHmi".LeftRobot.udiOdometer_X, udiOdometer_Z => "DB_ToHmi".LeftRobot.udiOdometer_Z, uiDistanceBeforeGreasingX => "DB_ToHmi".LeftRobot.uiDistanceBeforeGreasingX, uiDistanceBeforeGreasingZ => "DB_ToHmi".LeftRobot.uiDistanceBeforeGreasingZ, uiDiskUsed => "DB_ToHmi".LeftRobot.uiNbDiskUsed, uiRobotStatus => "DB_ToHmi".LeftRobot.uiRobotStatus, udiFaultTime => "DB_Exchange".LeftRobot.udiFaultTime, udiRunTime => "DB_Exchange".LeftRobot.udiRunTime, udiPauseTime => "DB_Exchange".LeftRobot.udiPauseTime, udiRobotPowerOnTime => "DB_Exchange".LeftRobot.udiRobotPowerOnTime, udiRobotDriveOnTime => "DB_Exchange".LeftRobot.udiRobotDriveOnTime, bInput100 => "DB_ToHmi".LeftRobot.IB_Input100, bInput101 => "DB_ToHmi".LeftRobot.IB_Input101, bInput102 => "DB_ToHmi".LeftRobot.IB_Input102, bInput103 => "DB_ToHmi".LeftRobot.IB_Input103, bInputFast90 => "DB_ToHmi".LeftRobot.IB_Fast90, bInputSafety500 => "DB_ToHmi".LeftRobot.IB_Safety500, bOutput100 => "DB_ToHmi".LeftRobot.OB_Output100, bOutput101 => "DB_ToHmi".LeftRobot.OB_Output101, bOutputSafety508 => "DB_ToHmi".LeftRobot.OB_Safety508, nInput600 => "DB_ToHmi".LeftRobot.IN_Input600, nInput602 => "DB_ToHmi".LeftRobot.IN_Input602, nInput604 => "DB_ToHmi".LeftRobot.IN_Input604, nInput606 => "DB_ToHmi".LeftRobot.IN_Input606, wFaultFerRobotic => "DB_ToHmi".Fault.wFerRoboticLeft, wFaultManageRobot => "DB_ToHmi".Fault.wManageRobotLeft, wFaultRobot => "DB_ToHmi".Fault.wRobotLeft, wFaultOther => "DB_ToHmi".Fault.wOtherLeft, wFaultVacuumValve => "DB_ToHmi".Fault.wVacuumValveLeft, wFaultFerRoboticManage => "DB_ToHmi".Fault.wFerRoboticManageLeft, wWarningDiskTrayEmpty => "DB_ToHmi".Warning.wWarnigLeft)
   END_RUNG
   // the same network as SCL:
   "iDB_CommLeftRobot"(InFromSlave := "IST_ReceiveLeft",   // "FB40_CommSlave"
                       xDryRun := "DB_FromHmi".xDryRun,
                       xResetGrafcet := "DB_FromHmi".LeftRobot.xResetGrafcet,
                       xAutoMode := "DB_Exchange".xAutoMode,
                       xSemiAutoMode := "DB_Exchange".xSemiAutoMode,
                       xMaintenanceMode := "DB_Exchange".xMaintenanceMode,
                       xReset := "DB_FromHmi".xResetFault,
                       xPulseSeconde := "Clock_1Hz",
                       xEnableStartRobot := "DB_FromHmi".xEnableStartLeftRobot,
                       xGlobalSafety := "DB_FromSafety".xGlobalSafetyLeft,
                       xCbsDoorAccessClosed := "DB_FromSafety".GateAccesCBS.State,
                       xAccessReq := "DB_Exchange".xStopRobotRequested,
                       xValideOperation := "DB_FromHmi".xValideOperation,
                       xValideFault := "DB_FromHmi".xValideFault,
                       xVaccumPumpRunning := "DB_FromSafety".VacuumPumpRunning.State,
                       xVacuumRunning := "DB_Exchange".xAuthorizationStartSanding,
                       xOtherRobotHasStarted := "DB_CommSlave".Right.xRobotHasStarted,
                       xOtherRobotFinished := "DB_CommSlave".Right.xRobotHasFinished,
                       xBothRobotFinished := "DB_CommSlave".Right.xBothSideFinished,
                       xReqChangePaper := "DB_FromHmi".LeftRobot.xReqChangeDisk,
                       xMaintStartProg := "DB_FromHmi".LeftRobot.xMaintStartProg,
                       xMaintStartMain := "DB_FromHmi".LeftRobot.xMaintStartMain,
                       usiRawMaterial := "DB_CurrentRecipe".WorkRecipe.RecipeRawMaterial,
                       uiServicePathNum := "DB_FromHmi".LeftRobot.uiServicePathNumber,
                       xParamManu := "DB_FromHmi".LeftRobot.ParamManu,
                       xCmdManuLockGimball := "DB_FromHmi".LeftRobot.xCmdManuLockGimball,
                       xCmdManuLockEccentric1 := "DB_FromHmi".LeftRobot.xCmdManuLockEccentric1,
                       xCmdManuLockEccentric2 := "DB_FromHmi".LeftRobot.xCmdManuLockEccentric2,
                       xCmdManuLockEccentric3 := "DB_FromHmi".LeftRobot.xCmdManuLockEccentric3,
                       xCmdManuEnableRotate := "DB_FromHmi".LeftRobot.xCmdManuEnableRotate,
                       xCmdManuRemoveConfig := "DB_FromHmi".LeftRobot.xCmdManuRemoveConfig,
                       xCmdManuPickupConfig := "DB_FromHmi".LeftRobot.xCmdManuPickupConfig,
                       xCmdManuFlatnessConfig := "DB_FromHmi".LeftRobot.xCmdManuFlatnessConfig,
                       xCmdManuOpenVacValve := "DB_FromHmi".LeftRobot.xCmdManuOpenVacValve,
                       xCmdManuCloseVaValve := "DB_FromHmi".LeftRobot.xCmdManuCloseVacValve,
                       xForceLubricationX := "DB_FromHmi".LeftRobot.xForceLubricationX,
                       xForceLubricationZ := "DB_FromHmi".LeftRobot.xForceLubricationZ,
                       xLightTest := "DB_FromHmi".xLightTest,
                       xStartRecipe := "DB_FromHmi".LeftRobot.xStartCycle,
                       xStopRecipe := "DB_FromHmi".LeftRobot.xStopCycle,
                       xCancelRecipe := "DB_FromHmi".LeftRobot.xCancelCycle,
                       xStartSanding := "DB_Exchange".xStartSanding,
                       xEndSanding := "DB_Exchange".xEndSanding,
                       xRobotUsed := "DB_Exchange".LeftRobot.xRobotUsed,
                       xStartPath := "DB_FromHmi".LeftRobot.xStartServicePath,
                       xStopPath := "DB_FromHmi".LeftRobot.xStopServicePath,
                       xCancelPath := "DB_FromHmi".LeftRobot.xCancelServicePath,
                       usiSandingType := "DB_CurrentRecipe".usiCurrentLayerType,
                       usiTrajNumber := "DB_CurrentRecipe".WorkRecipe.RecipeTrajNumber,
                       stFlatnessCtrlData := "DB_Exchange".stLeftRobotFlatnessCtrlData,
                       aListJobData := "DB_CurrentRecipe".WorkRecipe.RecipeLayerType.JobTableLeft,
                       OutToSlave => "OST_SendLeft",
                       xRobotInAuto => "DB_ToHmi".LeftRobot.xRobotInAuto,
                       xRobotInManu => "DB_ToHmi".LeftRobot.xRobotInManu,
                       xRobotInHome => "DB_ToHmi".xHomePositionR1,
                       xRobotReqReset => "DB_ToHmi".LeftRobot.xRobotReqReset,
                       xRobotStopped => "DB_Exchange".xLeftRobotStopped,
                       xWarningStart => "DB_Exchange".xStartUpWarningLeft,
                       xReqVacuum => "DB_Exchange".xLeftRobotStartVacuum,
                       xRecipeInProgress => "DB_ToHmi".LeftRobot.xRecipeInProgress,
                       xProductionRunning => "DB_Exchange".xProductionRunningRobot1,
                       xRobotHasStarted => "DB_CommSlave".Left.xRobotHasStarted,
                       xWaitOtherRobotFinished => "DB_CommSlave".Left.xRobotHasFinished,
                       xWaitBothRobotFinished => "DB_CommSlave".Left.xBothSideFinished,
                       xMagazineEmpty => "DB_ToHmi".LeftRobot.xMagazineEmpty,
                       xShowPopRemoveDisk => "DB_ToHmi".LeftRobot.xShowPopRemoveDisk,
                       xShowPopPickupDisk => "DB_ToHmi".LeftRobot.xShowPopPickupDisk,
                       xShowPopFlatnessFault => "DB_ToHmi".LeftRobot.xShowPopFlatnessFault,
                       uiJobDataNumber => "DB_ToHmi".LeftRobot.uiActualJobDataNumber,
                       xPathInProgress => "DB_ToHmi".LeftRobot.xPathInProgress,
                       xPathStopped => "DB_ToHmi".LeftRobot.xPathStopped,
                       xPathCancelled => "DB_ToHmi".LeftRobot.xPathCancelled,
                       xContactState => "DB_ToHmi".LeftRobot.xContactState,
                       xVacValveOpen => "DB_ToHmi".LeftRobot.xValveOpen,
                       xVacValveClosed => "DB_ToHmi".LeftRobot.xValveClosed,
                       nActualForce => "DB_ToHmi".LeftRobot.nActualForce,
                       uiSetSpeed => "DB_ToHmi".LeftRobot.uiSetSpeed,
                       uiRobotSpeed => "DB_ToHmi".LeftRobot.uiRobotSpeed,
                       uiPaperChangeDistance => "DB_ToHmi".LeftRobot.uiPaperChangeDistance,
                       rActualPosition => "DB_ToHmi".LeftRobot.rActualPosition,
                       xRangeFinderDetection => "DB_ToHmi".LeftRobot.xRangeFinderDetection,
                       uiRangeFinderValue => "DB_ToHmi".LeftRobot.uiRangeFinderValue,
                       uiCounterPulse_X => "DB_ToHmi".LeftRobot.uiCounterPulse_X,
                       uiCounterPulse_Z => "DB_ToHmi".LeftRobot.uiCounterPulse_Z,
                       uiGreaseFault_X => "DB_ToHmi".LeftRobot.uiGreaseFault_X,
                       uiGreaseFault_Z => "DB_ToHmi".LeftRobot.uiGreaseFault_Z,
                       uiDistanceSandingDisk => "DB_ToHmi".LeftRobot.uiDistanceSandingDisk,
                       uiActualRobotSpeed => "DB_ToHmi".LeftRobot.uiActualRobotSpeed,
                       udiOdometer_X => "DB_ToHmi".LeftRobot.udiOdometer_X,
                       udiOdometer_Z => "DB_ToHmi".LeftRobot.udiOdometer_Z,
                       uiDistanceBeforeGreasingX => "DB_ToHmi".LeftRobot.uiDistanceBeforeGreasingX,
                       uiDistanceBeforeGreasingZ => "DB_ToHmi".LeftRobot.uiDistanceBeforeGreasingZ,
                       uiDiskUsed => "DB_ToHmi".LeftRobot.uiNbDiskUsed,
                       uiRobotStatus => "DB_ToHmi".LeftRobot.uiRobotStatus,
                       udiFaultTime => "DB_Exchange".LeftRobot.udiFaultTime,
                       udiRunTime => "DB_Exchange".LeftRobot.udiRunTime,
                       udiPauseTime => "DB_Exchange".LeftRobot.udiPauseTime,
                       udiRobotPowerOnTime => "DB_Exchange".LeftRobot.udiRobotPowerOnTime,
                       udiRobotDriveOnTime => "DB_Exchange".LeftRobot.udiRobotDriveOnTime,
                       bInput100 => "DB_ToHmi".LeftRobot.IB_Input100,
                       bInput101 => "DB_ToHmi".LeftRobot.IB_Input101,
                       bInput102 => "DB_ToHmi".LeftRobot.IB_Input102,
                       bInput103 => "DB_ToHmi".LeftRobot.IB_Input103,
                       bInputFast90 => "DB_ToHmi".LeftRobot.IB_Fast90,
                       bInputSafety500 => "DB_ToHmi".LeftRobot.IB_Safety500,
                       bOutput100 => "DB_ToHmi".LeftRobot.OB_Output100,
                       bOutput101 => "DB_ToHmi".LeftRobot.OB_Output101,
                       bOutputSafety508 => "DB_ToHmi".LeftRobot.OB_Safety508,
                       nInput600 => "DB_ToHmi".LeftRobot.IN_Input600,
                       nInput602 => "DB_ToHmi".LeftRobot.IN_Input602,
                       nInput604 => "DB_ToHmi".LeftRobot.IN_Input604,
                       nInput606 => "DB_ToHmi".LeftRobot.IN_Input606,
                       wFaultFerRobotic => "DB_ToHmi".Fault.wFerRoboticLeft,
                       wFaultManageRobot => "DB_ToHmi".Fault.wManageRobotLeft,
                       wFaultRobot => "DB_ToHmi".Fault.wRobotLeft,
                       wFaultOther => "DB_ToHmi".Fault.wOtherLeft,
                       wFaultVacuumValve => "DB_ToHmi".Fault.wVacuumValveLeft,
                       wFaultFerRoboticManage => "DB_ToHmi".Fault.wFerRoboticManageLeft,
                       wWarningDiskTrayEmpty => "DB_ToHmi".Warning.wWarnigLeft);
END_REGION

REGION Network 2: Manage communication with Right PLC
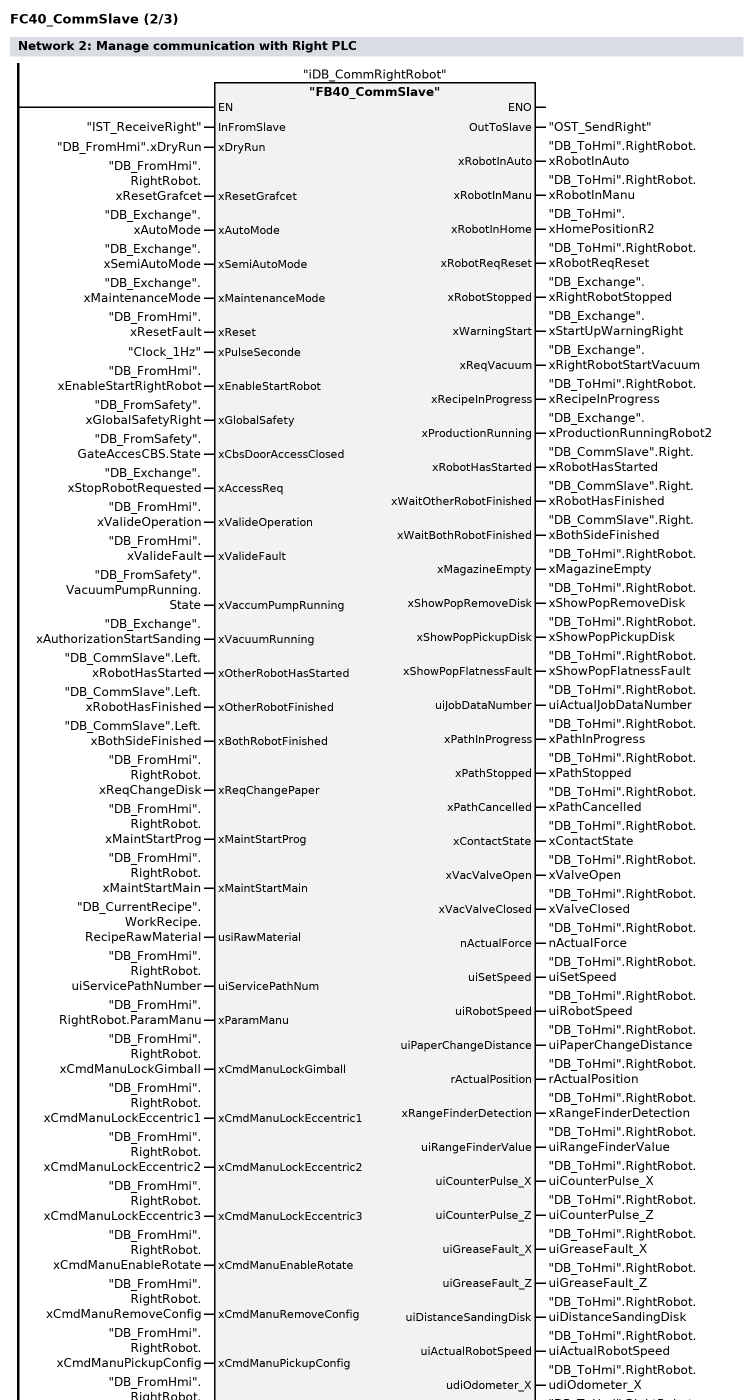
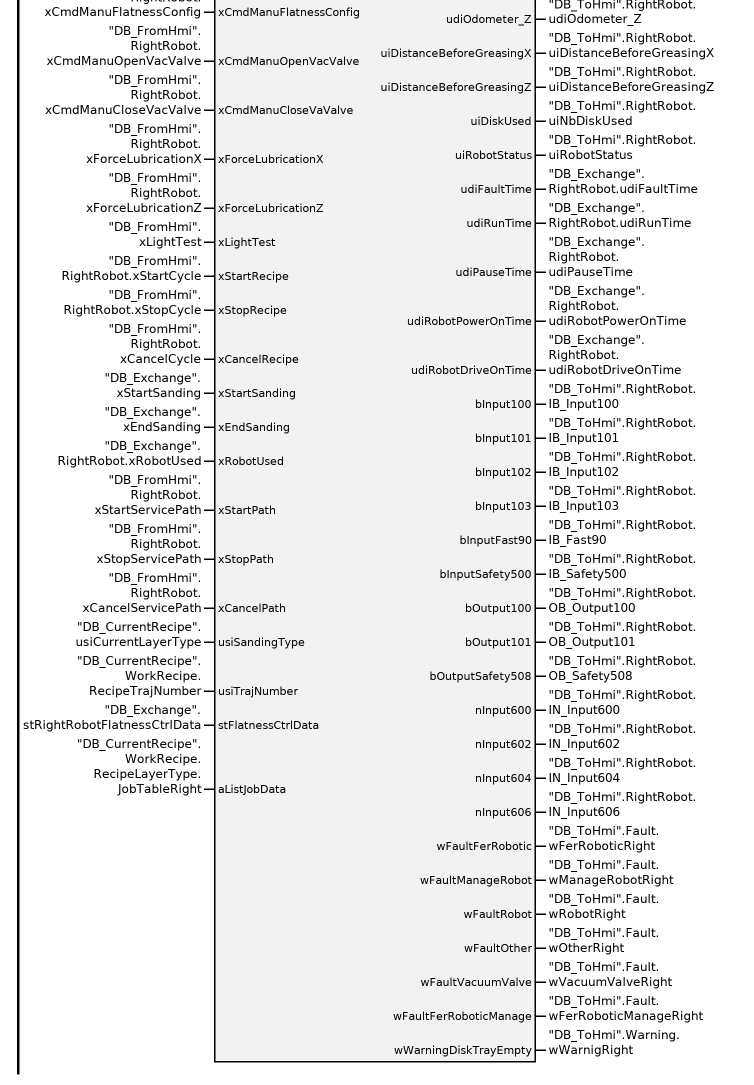
   RUNG wire#powerrail
      "iDB_CommRightRobot"(InFromSlave := "IST_ReceiveRight", xDryRun := "DB_FromHmi".xDryRun, xResetGrafcet := "DB_FromHmi".RightRobot.xResetGrafcet, xAutoMode := "DB_Exchange".xAutoMode, xSemiAutoMode := "DB_Exchange".xSemiAutoMode, xMaintenanceMode := "DB_Exchange".xMaintenanceMode, xReset := "DB_FromHmi".xResetFault, xPulseSeconde := "Clock_1Hz", xEnableStartRobot := "DB_FromHmi".xEnableStartRightRobot, xGlobalSafety := "DB_FromSafety".xGlobalSafetyRight, xCbsDoorAccessClosed := "DB_FromSafety".GateAccesCBS.State, xAccessReq := "DB_Exchange".xStopRobotRequested, xValideOperation := "DB_FromHmi".xValideOperation, xValideFault := "DB_FromHmi".xValideFault, xVaccumPumpRunning := "DB_FromSafety".VacuumPumpRunning.State, xVacuumRunning := "DB_Exchange".xAuthorizationStartSanding, xOtherRobotHasStarted := "DB_CommSlave".Left.xRobotHasStarted, xOtherRobotFinished := "DB_CommSlave".Left.xRobotHasFinished, xBothRobotFinished := "DB_CommSlave".Left.xBothSideFinished, xReqChangePaper := "DB_FromHmi".RightRobot.xReqChangeDisk, xMaintStartProg := "DB_FromHmi".RightRobot.xMaintStartProg, xMaintStartMain := "DB_FromHmi".RightRobot.xMaintStartMain, usiRawMaterial := "DB_CurrentRecipe".WorkRecipe.RecipeRawMaterial, uiServicePathNum := "DB_FromHmi".RightRobot.uiServicePathNumber, xParamManu := "DB_FromHmi".RightRobot.ParamManu, xCmdManuLockGimball := "DB_FromHmi".RightRobot.xCmdManuLockGimball, xCmdManuLockEccentric1 := "DB_FromHmi".RightRobot.xCmdManuLockEccentric1, xCmdManuLockEccentric2 := "DB_FromHmi".RightRobot.xCmdManuLockEccentric2, xCmdManuLockEccentric3 := "DB_FromHmi".RightRobot.xCmdManuLockEccentric3, xCmdManuEnableRotate := "DB_FromHmi".RightRobot.xCmdManuEnableRotate, xCmdManuRemoveConfig := "DB_FromHmi".RightRobot.xCmdManuRemoveConfig, xCmdManuPickupConfig := "DB_FromHmi".RightRobot.xCmdManuPickupConfig, xCmdManuFlatnessConfig := "DB_FromHmi".RightRobot.xCmdManuFlatnessConfig, xCmdManuOpenVacValve := "DB_FromHmi".RightRobot.xCmdManuOpenVacValve, xCmdManuCloseVaValve := "DB_FromHmi".RightRobot.xCmdManuCloseVacValve, xForceLubricationX := "DB_FromHmi".RightRobot.xForceLubricationX, xForceLubricationZ := "DB_FromHmi".RightRobot.xForceLubricationZ, xLightTest := "DB_FromHmi".xLightTest, xStartRecipe := "DB_FromHmi".RightRobot.xStartCycle, xStopRecipe := "DB_FromHmi".RightRobot.xStopCycle, xCancelRecipe := "DB_FromHmi".RightRobot.xCancelCycle, xStartSanding := "DB_Exchange".xStartSanding, xEndSanding := "DB_Exchange".xEndSanding, xRobotUsed := "DB_Exchange".RightRobot.xRobotUsed, xStartPath := "DB_FromHmi".RightRobot.xStartServicePath, xStopPath := "DB_FromHmi".RightRobot.xStopServicePath, xCancelPath := "DB_FromHmi".RightRobot.xCancelServicePath, usiSandingType := "DB_CurrentRecipe".usiCurrentLayerType, usiTrajNumber := "DB_CurrentRecipe".WorkRecipe.RecipeTrajNumber, stFlatnessCtrlData := "DB_Exchange".stRightRobotFlatnessCtrlData, aListJobData := "DB_CurrentRecipe".WorkRecipe.RecipeLayerType.JobTableRight, OutToSlave => "OST_SendRight", xRobotInAuto => "DB_ToHmi".RightRobot.xRobotInAuto, xRobotInManu => "DB_ToHmi".RightRobot.xRobotInManu, xRobotInHome => "DB_ToHmi".xHomePositionR2, xRobotReqReset => "DB_ToHmi".RightRobot.xRobotReqReset, xRobotStopped => "DB_Exchange".xRightRobotStopped, xWarningStart => "DB_Exchange".xStartUpWarningRight, xReqVacuum => "DB_Exchange".xRightRobotStartVacuum, xRecipeInProgress => "DB_ToHmi".RightRobot.xRecipeInProgress, xProductionRunning => "DB_Exchange".xProductionRunningRobot2, xRobotHasStarted => "DB_CommSlave".Right.xRobotHasStarted, xWaitOtherRobotFinished => "DB_CommSlave".Right.xRobotHasFinished, xWaitBothRobotFinished => "DB_CommSlave".Right.xBothSideFinished, xMagazineEmpty => "DB_ToHmi".RightRobot.xMagazineEmpty, xShowPopRemoveDisk => "DB_ToHmi".RightRobot.xShowPopRemoveDisk, xShowPopPickupDisk => "DB_ToHmi".RightRobot.xShowPopPickupDisk, xShowPopFlatnessFault => "DB_ToHmi".RightRobot.xShowPopFlatnessFault, uiJobDataNumber => "DB_ToHmi".RightRobot.uiActualJobDataNumber, xPathInProgress => "DB_ToHmi".RightRobot.xPathInProgress, xPathStopped => "DB_ToHmi".RightRobot.xPathStopped, xPathCancelled => "DB_ToHmi".RightRobot.xPathCancelled, xContactState => "DB_ToHmi".RightRobot.xContactState, xVacValveOpen => "DB_ToHmi".RightRobot.xValveOpen, xVacValveClosed => "DB_ToHmi".RightRobot.xValveClosed, nActualForce => "DB_ToHmi".RightRobot.nActualForce, uiSetSpeed => "DB_ToHmi".RightRobot.uiSetSpeed, uiRobotSpeed => "DB_ToHmi".RightRobot.uiRobotSpeed, uiPaperChangeDistance => "DB_ToHmi".RightRobot.uiPaperChangeDistance, rActualPosition => "DB_ToHmi".RightRobot.rActualPosition, xRangeFinderDetection => "DB_ToHmi".RightRobot.xRangeFinderDetection, uiRangeFinderValue => "DB_ToHmi".RightRobot.uiRangeFinderValue, uiCounterPulse_X => "DB_ToHmi".RightRobot.uiCounterPulse_X, uiCounterPulse_Z => "DB_ToHmi".RightRobot.uiCounterPulse_Z, uiGreaseFault_X => "DB_ToHmi".RightRobot.uiGreaseFault_X, uiGreaseFault_Z => "DB_ToHmi".RightRobot.uiGreaseFault_Z, uiDistanceSandingDisk => "DB_ToHmi".RightRobot.uiDistanceSandingDisk, uiActualRobotSpeed => "DB_ToHmi".RightRobot.uiActualRobotSpeed, udiOdometer_X => "DB_ToHmi".RightRobot.udiOdometer_X, udiOdometer_Z => "DB_ToHmi".RightRobot.udiOdometer_Z, uiDistanceBeforeGreasingX => "DB_ToHmi".RightRobot.uiDistanceBeforeGreasingX, uiDistanceBeforeGreasingZ => "DB_ToHmi".RightRobot.uiDistanceBeforeGreasingZ, uiDiskUsed => "DB_ToHmi".RightRobot.uiNbDiskUsed, uiRobotStatus => "DB_ToHmi".RightRobot.uiRobotStatus, udiFaultTime => "DB_Exchange".RightRobot.udiFaultTime, udiRunTime => "DB_Exchange".RightRobot.udiRunTime, udiPauseTime => "DB_Exchange".RightRobot.udiPauseTime, udiRobotPowerOnTime => "DB_Exchange".RightRobot.udiRobotPowerOnTime, udiRobotDriveOnTime => "DB_Exchange".RightRobot.udiRobotDriveOnTime, bInput100 => "DB_ToHmi".RightRobot.IB_Input100, bInput101 => "DB_ToHmi".RightRobot.IB_Input101, bInput102 => "DB_ToHmi".RightRobot.IB_Input102, bInput103 => "DB_ToHmi".RightRobot.IB_Input103, bInputFast90 => "DB_ToHmi".RightRobot.IB_Fast90, bInputSafety500 => "DB_ToHmi".RightRobot.IB_Safety500, bOutput100 => "DB_ToHmi".RightRobot.OB_Output100, bOutput101 => "DB_ToHmi".RightRobot.OB_Output101, bOutputSafety508 => "DB_ToHmi".RightRobot.OB_Safety508, nInput600 => "DB_ToHmi".RightRobot.IN_Input600, nInput602 => "DB_ToHmi".RightRobot.IN_Input602, nInput604 => "DB_ToHmi".RightRobot.IN_Input604, nInput606 => "DB_ToHmi".RightRobot.IN_Input606, wFaultFerRobotic => "DB_ToHmi".Fault.wFerRoboticRight, wFaultManageRobot => "DB_ToHmi".Fault.wManageRobotRight, wFaultRobot => "DB_ToHmi".Fault.wRobotRight, wFaultOther => "DB_ToHmi".Fault.wOtherRight, wFaultVacuumValve => "DB_ToHmi".Fault.wVacuumValveRight, wFaultFerRoboticManage => "DB_ToHmi".Fault.wFerRoboticManageRight, wWarningDiskTrayEmpty => "DB_ToHmi".Warning.wWarnigRight)
   END_RUNG
   // the same network as SCL:
   "iDB_CommRightRobot"(InFromSlave := "IST_ReceiveRight",   // "FB40_CommSlave"
                        xDryRun := "DB_FromHmi".xDryRun,
                        xResetGrafcet := "DB_FromHmi".RightRobot.xResetGrafcet,
                        xAutoMode := "DB_Exchange".xAutoMode,
                        xSemiAutoMode := "DB_Exchange".xSemiAutoMode,
                        xMaintenanceMode := "DB_Exchange".xMaintenanceMode,
                        xReset := "DB_FromHmi".xResetFault,
                        xPulseSeconde := "Clock_1Hz",
                        xEnableStartRobot := "DB_FromHmi".xEnableStartRightRobot,
                        xGlobalSafety := "DB_FromSafety".xGlobalSafetyRight,
                        xCbsDoorAccessClosed := "DB_FromSafety".GateAccesCBS.State,
                        xAccessReq := "DB_Exchange".xStopRobotRequested,
                        xValideOperation := "DB_FromHmi".xValideOperation,
                        xValideFault := "DB_FromHmi".xValideFault,
                        xVaccumPumpRunning := "DB_FromSafety".VacuumPumpRunning.State,
                        xVacuumRunning := "DB_Exchange".xAuthorizationStartSanding,
                        xOtherRobotHasStarted := "DB_CommSlave".Left.xRobotHasStarted,
                        xOtherRobotFinished := "DB_CommSlave".Left.xRobotHasFinished,
                        xBothRobotFinished := "DB_CommSlave".Left.xBothSideFinished,
                        xReqChangePaper := "DB_FromHmi".RightRobot.xReqChangeDisk,
                        xMaintStartProg := "DB_FromHmi".RightRobot.xMaintStartProg,
                        xMaintStartMain := "DB_FromHmi".RightRobot.xMaintStartMain,
                        usiRawMaterial := "DB_CurrentRecipe".WorkRecipe.RecipeRawMaterial,
                        uiServicePathNum := "DB_FromHmi".RightRobot.uiServicePathNumber,
                        xParamManu := "DB_FromHmi".RightRobot.ParamManu,
                        xCmdManuLockGimball := "DB_FromHmi".RightRobot.xCmdManuLockGimball,
                        xCmdManuLockEccentric1 := "DB_FromHmi".RightRobot.xCmdManuLockEccentric1,
                        xCmdManuLockEccentric2 := "DB_FromHmi".RightRobot.xCmdManuLockEccentric2,
                        xCmdManuLockEccentric3 := "DB_FromHmi".RightRobot.xCmdManuLockEccentric3,
                        xCmdManuEnableRotate := "DB_FromHmi".RightRobot.xCmdManuEnableRotate,
                        xCmdManuRemoveConfig := "DB_FromHmi".RightRobot.xCmdManuRemoveConfig,
                        xCmdManuPickupConfig := "DB_FromHmi".RightRobot.xCmdManuPickupConfig,
                        xCmdManuFlatnessConfig := "DB_FromHmi".RightRobot.xCmdManuFlatnessConfig,
                        xCmdManuOpenVacValve := "DB_FromHmi".RightRobot.xCmdManuOpenVacValve,
                        xCmdManuCloseVaValve := "DB_FromHmi".RightRobot.xCmdManuCloseVacValve,
                        xForceLubricationX := "DB_FromHmi".RightRobot.xForceLubricationX,
                        xForceLubricationZ := "DB_FromHmi".RightRobot.xForceLubricationZ,
                        xLightTest := "DB_FromHmi".xLightTest,
                        xStartRecipe := "DB_FromHmi".RightRobot.xStartCycle,
                        xStopRecipe := "DB_FromHmi".RightRobot.xStopCycle,
                        xCancelRecipe := "DB_FromHmi".RightRobot.xCancelCycle,
                        xStartSanding := "DB_Exchange".xStartSanding,
                        xEndSanding := "DB_Exchange".xEndSanding,
                        xRobotUsed := "DB_Exchange".RightRobot.xRobotUsed,
                        xStartPath := "DB_FromHmi".RightRobot.xStartServicePath,
                        xStopPath := "DB_FromHmi".RightRobot.xStopServicePath,
                        xCancelPath := "DB_FromHmi".RightRobot.xCancelServicePath,
                        usiSandingType := "DB_CurrentRecipe".usiCurrentLayerType,
                        usiTrajNumber := "DB_CurrentRecipe".WorkRecipe.RecipeTrajNumber,
                        stFlatnessCtrlData := "DB_Exchange".stRightRobotFlatnessCtrlData,
                        aListJobData := "DB_CurrentRecipe".WorkRecipe.RecipeLayerType.JobTableRight,
                        OutToSlave => "OST_SendRight",
                        xRobotInAuto => "DB_ToHmi".RightRobot.xRobotInAuto,
                        xRobotInManu => "DB_ToHmi".RightRobot.xRobotInManu,
                        xRobotInHome => "DB_ToHmi".xHomePositionR2,
                        xRobotReqReset => "DB_ToHmi".RightRobot.xRobotReqReset,
                        xRobotStopped => "DB_Exchange".xRightRobotStopped,
                        xWarningStart => "DB_Exchange".xStartUpWarningRight,
                        xReqVacuum => "DB_Exchange".xRightRobotStartVacuum,
                        xRecipeInProgress => "DB_ToHmi".RightRobot.xRecipeInProgress,
                        xProductionRunning => "DB_Exchange".xProductionRunningRobot2,
                        xRobotHasStarted => "DB_CommSlave".Right.xRobotHasStarted,
                        xWaitOtherRobotFinished => "DB_CommSlave".Right.xRobotHasFinished,
                        xWaitBothRobotFinished => "DB_CommSlave".Right.xBothSideFinished,
                        xMagazineEmpty => "DB_ToHmi".RightRobot.xMagazineEmpty,
                        xShowPopRemoveDisk => "DB_ToHmi".RightRobot.xShowPopRemoveDisk,
                        xShowPopPickupDisk => "DB_ToHmi".RightRobot.xShowPopPickupDisk,
                        xShowPopFlatnessFault => "DB_ToHmi".RightRobot.xShowPopFlatnessFault,
                        uiJobDataNumber => "DB_ToHmi".RightRobot.uiActualJobDataNumber,
                        xPathInProgress => "DB_ToHmi".RightRobot.xPathInProgress,
                        xPathStopped => "DB_ToHmi".RightRobot.xPathStopped,
                        xPathCancelled => "DB_ToHmi".RightRobot.xPathCancelled,
                        xContactState => "DB_ToHmi".RightRobot.xContactState,
                        xVacValveOpen => "DB_ToHmi".RightRobot.xValveOpen,
                        xVacValveClosed => "DB_ToHmi".RightRobot.xValveClosed,
                        nActualForce => "DB_ToHmi".RightRobot.nActualForce,
                        uiSetSpeed => "DB_ToHmi".RightRobot.uiSetSpeed,
                        uiRobotSpeed => "DB_ToHmi".RightRobot.uiRobotSpeed,
                        uiPaperChangeDistance => "DB_ToHmi".RightRobot.uiPaperChangeDistance,
                        rActualPosition => "DB_ToHmi".RightRobot.rActualPosition,
                        xRangeFinderDetection => "DB_ToHmi".RightRobot.xRangeFinderDetection,
                        uiRangeFinderValue => "DB_ToHmi".RightRobot.uiRangeFinderValue,
                        uiCounterPulse_X => "DB_ToHmi".RightRobot.uiCounterPulse_X,
                        uiCounterPulse_Z => "DB_ToHmi".RightRobot.uiCounterPulse_Z,
                        uiGreaseFault_X => "DB_ToHmi".RightRobot.uiGreaseFault_X,
                        uiGreaseFault_Z => "DB_ToHmi".RightRobot.uiGreaseFault_Z,
                        uiDistanceSandingDisk => "DB_ToHmi".RightRobot.uiDistanceSandingDisk,
                        uiActualRobotSpeed => "DB_ToHmi".RightRobot.uiActualRobotSpeed,
                        udiOdometer_X => "DB_ToHmi".RightRobot.udiOdometer_X,
                        udiOdometer_Z => "DB_ToHmi".RightRobot.udiOdometer_Z,
                        uiDistanceBeforeGreasingX => "DB_ToHmi".RightRobot.uiDistanceBeforeGreasingX,
                        uiDistanceBeforeGreasingZ => "DB_ToHmi".RightRobot.uiDistanceBeforeGreasingZ,
                        uiDiskUsed => "DB_ToHmi".RightRobot.uiNbDiskUsed,
                        uiRobotStatus => "DB_ToHmi".RightRobot.uiRobotStatus,
                        udiFaultTime => "DB_Exchange".RightRobot.udiFaultTime,
                        udiRunTime => "DB_Exchange".RightRobot.udiRunTime,
                        udiPauseTime => "DB_Exchange".RightRobot.udiPauseTime,
                        udiRobotPowerOnTime => "DB_Exchange".RightRobot.udiRobotPowerOnTime,
                        udiRobotDriveOnTime => "DB_Exchange".RightRobot.udiRobotDriveOnTime,
                        bInput100 => "DB_ToHmi".RightRobot.IB_Input100,
                        bInput101 => "DB_ToHmi".RightRobot.IB_Input101,
                        bInput102 => "DB_ToHmi".RightRobot.IB_Input102,
                        bInput103 => "DB_ToHmi".RightRobot.IB_Input103,
                        bInputFast90 => "DB_ToHmi".RightRobot.IB_Fast90,
                        bInputSafety500 => "DB_ToHmi".RightRobot.IB_Safety500,
                        bOutput100 => "DB_ToHmi".RightRobot.OB_Output100,
                        bOutput101 => "DB_ToHmi".RightRobot.OB_Output101,
                        bOutputSafety508 => "DB_ToHmi".RightRobot.OB_Safety508,
                        nInput600 => "DB_ToHmi".RightRobot.IN_Input600,
                        nInput602 => "DB_ToHmi".RightRobot.IN_Input602,
                        nInput604 => "DB_ToHmi".RightRobot.IN_Input604,
                        nInput606 => "DB_ToHmi".RightRobot.IN_Input606,
                        wFaultFerRobotic => "DB_ToHmi".Fault.wFerRoboticRight,
                        wFaultManageRobot => "DB_ToHmi".Fault.wManageRobotRight,
                        wFaultRobot => "DB_ToHmi".Fault.wRobotRight,
                        wFaultOther => "DB_ToHmi".Fault.wOtherRight,
                        wFaultVacuumValve => "DB_ToHmi".Fault.wVacuumValveRight,
                        wFaultFerRoboticManage => "DB_ToHmi".Fault.wFerRoboticManageRight,
                        wWarningDiskTrayEmpty => "DB_ToHmi".Warning.wWarnigRight);
END_REGION

REGION Network 3: Sanding process is in progress
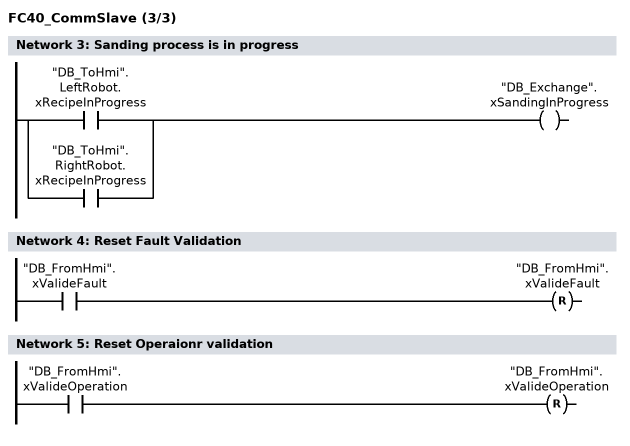
   RUNG wire#powerrail
      Contact( "DB_ToHmi".LeftRobot.xRecipeInProgress )
      wire#w1
      Coil( "DB_Exchange".xSandingInProgress )
   END_RUNG
   RUNG wire#powerrail
      Contact( "DB_ToHmi".RightRobot.xRecipeInProgress )
   END_RUNG wire#w1
   // the same network as SCL:
   "DB_Exchange".xSandingInProgress := "DB_ToHmi".LeftRobot.xRecipeInProgress OR "DB_ToHmi".RightRobot.xRecipeInProgress;
END_REGION

REGION Network 4: Reset Fault Validation
   RUNG wire#powerrail
      Contact( "DB_FromHmi".xValideFault )
      R_Coil( "DB_FromHmi".xValideFault )
   END_RUNG
   // the same network as SCL:
   IF "DB_FromHmi".xValideFault THEN "DB_FromHmi".xValideFault := FALSE; END_IF;
END_REGION

REGION Network 5: Reset Operaionr validation
   RUNG wire#powerrail
      Contact( "DB_FromHmi".xValideOperation )
      R_Coil( "DB_FromHmi".xValideOperation )
   END_RUNG
   // the same network as SCL:
   IF "DB_FromHmi".xValideOperation THEN "DB_FromHmi".xValideOperation := FALSE; END_IF;
END_REGION
END_FUNCTION

